   S700_1_WELD_BUFF_DATA5.RBT23_WELD_COUNT := W#16#0;
   S700_1_WELD_BUFF_DATA5.RBT24_BT_CODE_NO := W#16#0;
   S700_1_WELD_BUFF_DATA5.RBT24_WELD_COUNT := W#16#0;
   S700_1_WELD_BUFF_DATA5.WELD_DETERMINES_RESULT := W#16#0;
   S700_1_WELD_BUFF_DATA5.WELD_CHECK_SUM := W#16#0;
   S700_1_WELD_BUFF_DATA5.SPARE1 := W#16#0;
   S700_1_WELD_BUFF_DATA6.STATION_MAIN := W#16#0;
   S700_1_WELD_BUFF_DATA6.DISTINCTION_LH_RH := W#16#0;
   S700_1_WELD_BUFF_DATA6.STAION_NUMBER := W#16#0;
   S700_1_WELD_BUFF_DATA6.VIN_NUMBER1 := W#16#0;
   S700_1_WELD_BUFF_DATA6.VIN_NUMBER2 := W#16#0;
   S700_1_WELD_BUFF_DATA6.VIN_NUMBER3 := W#16#0;
   S700_1_WELD_BUFF_DATA6.VIN_NUMBER4 := W#16#0;
   S700_1_WELD_BUFF_DATA6.SEQ_NUMBER1 := W#16#0;
   S700_1_WELD_BUFF_DATA6.SEQ_NUMBER2 := W#16#0;
   S700_1_WELD_BUFF_DATA6.RBT1_BT_CODE_NO := W#16#0;
   S700_1_WELD_BUFF_DATA6.RBT1_WELD_COUNT := W#16#0;
   S700_1_WELD_BUFF_DATA6.RBT2_BT_CODE_NO := W#16#0;
   S700_1_WELD_BUFF_DATA6.RBT2_WELD_COUNT := W#16#0;
   S700_1_WELD_BUFF_DATA6.RBT3_BT_CODE_NO := W#16#0;
   S700_1_WELD_BUFF_DATA6.RBT3_WELD_COUNT := W#16#0;
   S700_1_WELD_BUFF_DATA6.RBT4_BT_CODE_NO := W#16#0;
   S700_1_WELD_BUFF_DATA6.RBT4_WELD_COUNT := W#16#0;
   S700_1_WELD_BUFF_DATA6.RBT5_BT_CODE_NO := W#16#0;
   S700_1_WELD_BUFF_DATA6.RBT5_WELD_COUNT := W#16#0;
   S700_1_WELD_BUFF_DATA6.RBT6_BT_CODE_NO := W#16#0;
   S700_1_WELD_BUFF_DATA6.RBT6_WELD_COUNT := W#16#0;
   S700_1_WELD_BUFF_DATA6.RBT7_BT_CODE_NO := W#16#0;
   S700_1_WELD_BUFF_DATA6.RBT7_WELD_COUNT := W#16#0;
   S700_1_WELD_BUFF_DATA6.RBT8_BT_CODE_NO := W#16#0;
   S700_1_WELD_BUFF_DATA6.RBT8_WELD_COUNT := W#16#0;
   S700_1_WELD_BUFF_DATA6.RBT9_BT_CODE_NO := W#16#0;
   S700_1_WELD_BUFF_DATA6.RBT9_WELD_COUNT := W#16#0;
   S700_1_WELD_BUFF_DATA6.RBT10_BT_CODE_NO := W#16#0;
   S700_1_WELD_BUFF_DATA6.RBT10_WELD_COUNT := W#16#0;
   S700_1_WELD_BUFF_DATA6.RBT11_BT_CODE_NO := W#16#0;
   S700_1_WELD_BUFF_DATA6.RBT11_WELD_COUNT := W#16#0;
   S700_1_WELD_BUFF_DATA6.RBT12_BT_CODE_NO := W#16#0;
   S700_1_WELD_BUFF_DATA6.RBT12_WELD_COUNT := W#16#0;
   S700_1_WELD_BUFF_DATA6.RBT13_BT_CODE_NO := W#16#0;
   S700_1_WELD_BUFF_DATA6.RBT13_WELD_COUNT := W#16#0;
   S700_1_WELD_BUFF_DATA6.RBT14_BT_CODE_NO := W#16#0;
   S700_1_WELD_BUFF_DATA6.RBT14_WELD_COUNT := W#16#0;
   S700_1_WELD_BUFF_DATA6.RBT15_BT_CODE_NO := W#16#0;
   S700_1_WELD_BUFF_DATA6.RBT15_WELD_COUNT := W#16#0;
   S700_1_WELD_BUFF_DATA6.RBT16_BT_CODE_NO := W#16#0;
   S700_1_WELD_BUFF_DATA6.RBT16_WELD_COUNT := W#16#0;
   S700_1_WELD_BUFF_DATA6.RBT17_BT_CODE_NO := W#16#0;
   S700_1_WELD_BUFF_DATA6.RBT17_WELD_COUNT := W#16#0;
   S700_1_WELD_BUFF_DATA6.RBT18_BT_CODE_NO := W#16#0;
   S700_1_WELD_BUFF_DATA6.RBT18_WELD_COUNT := W#16#0;
   S700_1_WELD_BUFF_DATA6.RBT19_BT_CODE_NO := W#16#0;
   S700_1_WELD_BUFF_DATA6.RBT19_WELD_COUNT := W#16#0;
   S700_1_WELD_BUFF_DATA6.RBT20_BT_CODE_NO := W#16#0;
   S700_1_WELD_BUFF_DATA6.RBT20_WELD_COUNT := W#16#0;
   S700_1_WELD_BUFF_DATA6.RBT21_BT_CODE_NO := W#16#0;
   S700_1_WELD_BUFF_DATA6.RBT21_WELD_COUNT := W#16#0;
   S700_1_WELD_BUFF_DATA6.RBT22_BT_CODE_NO := W#16#0;
   S700_1_WELD_BUFF_DATA6.RBT22_WELD_COUNT := W#16#0;
   S700_1_WELD_BUFF_DATA6.RBT23_BT_CODE_NO := W#16#0;
   S700_1_WELD_BUFF_DATA6.RBT23_WELD_COUNT := W#16#0;
   S700_1_WELD_BUFF_DATA6.RBT24_BT_CODE_NO := W#16#0;
   S700_1_WELD_BUFF_DATA6.RBT24_WELD_COUNT := W#16#0;
   S700_1_WELD_BUFF_DATA6.WELD_DETERMINES_RESULT := W#16#0;
   S700_1_WELD_BUFF_DATA6.WELD_CHECK_SUM := W#16#0;
   S700_1_WELD_BUFF_DATA6.SPARE1 := W#16#0;
   S700_1_WELD_BUFF_DATA7.STATION_MAIN := W#16#0;
   S700_1_WELD_BUFF_DATA7.DISTINCTION_LH_RH := W#16#0;
   S700_1_WELD_BUFF_DATA7.STAION_NUMBER := W#16#0;
   S700_1_WELD_BUFF_DATA7.VIN_NUMBER1 := W#16#0;
   S700_1_WELD_BUFF_DATA7.VIN_NUMBER2 := W#16#0;
   S700_1_WELD_BUFF_DATA7.VIN_NUMBER3 := W#16#0;
   S700_1_WELD_BUFF_DATA7.VIN_NUMBER4 := W#16#0;
   S700_1_WELD_BUFF_DATA7.SEQ_NUMBER1 := W#16#0;
   S700_1_WELD_BUFF_DATA7.SEQ_NUMBER2 := W#16#0;
   S700_1_WELD_BUFF_DATA7.RBT1_BT_CODE_NO := W#16#0;
   S700_1_WELD_BUFF_DATA7.RBT1_WELD_COUNT := W#16#0;
   S700_1_WELD_BUFF_DATA7.RBT2_BT_CODE_NO := W#16#0;
   S700_1_WELD_BUFF_DATA7.RBT2_WELD_COUNT := W#16#0;
   S700_1_WELD_BUFF_DATA7.RBT3_BT_CODE_NO := W#16#0;
   S700_1_WELD_BUFF_DATA7.RBT3_WELD_COUNT := W#16#0;
   S700_1_WELD_BUFF_DATA7.RBT4_BT_CODE_NO := W#16#0;
   S700_1_WELD_BUFF_DATA7.RBT4_WELD_COUNT := W#16#0;
   S700_1_WELD_BUFF_DATA7.RBT5_BT_CODE_NO := W#16#0;
   S700_1_WELD_BUFF_DATA7.RBT5_WELD_COUNT := W#16#0;
   S700_1_WELD_BUFF_DATA7.RBT6_BT_CODE_NO := W#16#0;
   S700_1_WELD_BUFF_DATA7.RBT6_WELD_COUNT := W#16#0;
   S700_1_WELD_BUFF_DATA7.RBT7_BT_CODE_NO := W#16#0;
   S700_1_WELD_BUFF_DATA7.RBT7_WELD_COUNT := W#16#0;
   S700_1_WELD_BUFF_DATA7.RBT8_BT_CODE_NO := W#16#0;
   S700_1_WELD_BUFF_DATA7.RBT8_WELD_COUNT := W#16#0;
   S700_1_WELD_BUFF_DATA7.RBT9_BT_CODE_NO := W#16#0;
   S700_1_WELD_BUFF_DATA7.RBT9_WELD_COUNT := W#16#0;
   S700_1_WELD_BUFF_DATA7.RBT10_BT_CODE_NO := W#16#0;
   S700_1_WELD_BUFF_DATA7.RBT10_WELD_COUNT := W#16#0;
   S700_1_WELD_BUFF_DATA7.RBT11_BT_CODE_NO := W#16#0;
   S700_1_WELD_BUFF_DATA7.RBT11_WELD_COUNT := W#16#0;
   S700_1_WELD_BUFF_DATA7.RBT12_BT_CODE_NO := W#16#0;
   S700_1_WELD_BUFF_DATA7.RBT12_WELD_COUNT := W#16#0;
   S700_1_WELD_BUFF_DATA7.RBT13_BT_CODE_NO := W#16#0;
   S700_1_WELD_BUFF_DATA7.RBT13_WELD_COUNT := W#16#0;
   S700_1_WELD_BUFF_DATA7.RBT14_BT_CODE_NO := W#16#0;
   S700_1_WELD_BUFF_DATA7.RBT14_WELD_COUNT := W#16#0;
   S700_1_WELD_BUFF_DATA7.RBT15_BT_CODE_NO := W#16#0;
   S700_1_WELD_BUFF_DATA7.RBT15_WELD_COUNT := W#16#0;
   S700_1_WELD_BUFF_DATA7.RBT16_BT_CODE_NO := W#16#0;
   S700_1_WELD_BUFF_DATA7.RBT16_WELD_COUNT := W#16#0;
   S700_1_WELD_BUFF_DATA7.RBT17_BT_CODE_NO := W#16#0;
   S700_1_WELD_BUFF_DATA7.RBT17_WELD_COUNT := W#16#0;
   S700_1_WELD_BUFF_DATA7.RBT18_BT_CODE_NO := W#16#0;
   S700_1_WELD_BUFF_DATA7.RBT18_WELD_COUNT := W#16#0;
   S700_1_WELD_BUFF_DATA7.RBT19_BT_CODE_NO := W#16#0;
   S700_1_WELD_BUFF_DATA7.RBT19_WELD_COUNT := W#16#0;
   S700_1_WELD_BUFF_DATA7.RBT20_BT_CODE_NO := W#16#0;
   S700_1_WELD_BUFF_DATA7.RBT20_WELD_COUNT := W#16#0;
   S700_1_WELD_BUFF_DATA7.RBT21_BT_CODE_NO := W#16#0;
   S700_1_WELD_BUFF_DATA7.RBT21_WELD_COUNT := W#16#0;
   S700_1_WELD_BUFF_DATA7.RBT22_BT_CODE_NO := W#16#0;
   S700_1_WELD_BUFF_DATA7.RBT22_WELD_COUNT := W#16#0;
   S700_1_WELD_BUFF_DATA7.RBT23_BT_CODE_NO := W#16#0;
   S700_1_WELD_BUFF_DATA7.RBT23_WELD_COUNT := W#16#0;
   S700_1_WELD_BUFF_DATA7.RBT24_BT_CODE_NO := W#16#0;
   S700_1_WELD_BUFF_DATA7.RBT24_WELD_COUNT := W#16#0;
   S700_1_WELD_BUFF_DATA7.WELD_DETERMINES_RESULT := W#16#0;
   S700_1_WELD_BUFF_DATA7.WELD_CHECK_SUM := W#16#0;
   S700_1_WELD_BUFF_DATA7.SPARE1 := W#16#0;
   S700_1_WELD_BUFF_DATA8.STATION_MAIN := W#16#0;
   S700_1_WELD_BUFF_DATA8.DISTINCTION_LH_RH := W#16#0;
   S700_1_WELD_BUFF_DATA8.STAION_NUMBER := W#16#0;
   S700_1_WELD_BUFF_DATA8.VIN_NUMBER1 := W#16#0;
   S700_1_WELD_BUFF_DATA8.VIN_NUMBER2 := W#16#0;
   S700_1_WELD_BUFF_DATA8.VIN_NUMBER3 := W#16#0;
   S700_1_WELD_BUFF_DATA8.VIN_NUMBER4 := W#16#0;
   S700_1_WELD_BUFF_DATA8.SEQ_NUMBER1 := W#16#0;
   S700_1_WELD_BUFF_DATA8.SEQ_NUMBER2 := W#16#0;
   S700_1_WELD_BUFF_DATA8.RBT1_BT_CODE_NO := W#16#0;
   S700_1_WELD_BUFF_DATA8.RBT1_WELD_COUNT := W#16#0;
   S700_1_WELD_BUFF_DATA8.RBT2_BT_CODE_NO := W#16#0;
   S700_1_WELD_BUFF_DATA8.RBT2_WELD_COUNT := W#16#0;
   S700_1_WELD_BUFF_DATA8.RBT3_BT_CODE_NO := W#16#0;
   S700_1_WELD_BUFF_DATA8.RBT3_WELD_COUNT := W#16#0;
   S700_1_WELD_BUFF_DATA8.RBT4_BT_CODE_NO := W#16#0;
   S700_1_WELD_BUFF_DATA8.RBT4_WELD_COUNT := W#16#0;
   S700_1_WELD_BUFF_DATA8.RBT5_BT_CODE_NO := W#16#0;
   S700_1_WELD_BUFF_DATA8.RBT5_WELD_COUNT := W#16#0;
   S700_1_WELD_BUFF_DATA8.RBT6_BT_CODE_NO := W#16#0;
   S700_1_WELD_BUFF_DATA8.RBT6_WELD_COUNT := W#16#0;
   S700_1_WELD_BUFF_DATA8.RBT7_BT_CODE_NO := W#16#0;
   S700_1_WELD_BUFF_DATA8.RBT7_WELD_COUNT := W#16#0;
   S700_1_WELD_BUFF_DATA8.RBT8_BT_CODE_NO := W#16#0;
   S700_1_WELD_BUFF_DATA8.RBT8_WELD_COUNT := W#16#0;
   S700_1_WELD_BUFF_DATA8.RBT9_BT_CODE_NO := W#16#0;
   S700_1_WELD_BUFF_DATA8.RBT9_WELD_COUNT := W#16#0;
   S700_1_WELD_BUFF_DATA8.RBT10_BT_CODE_NO := W#16#0;
   S700_1_WELD_BUFF_DATA8.RBT10_WELD_COUNT := W#16#0;
   S700_1_WELD_BUFF_DATA8.RBT11_BT_CODE_NO := W#16#0;
   S700_1_WELD_BUFF_DATA8.RBT11_WELD_COUNT := W#16#0;
   S700_1_WELD_BUFF_DATA8.RBT12_BT_CODE_NO := W#16#0;
   S700_1_WELD_BUFF_DATA8.RBT12_WELD_COUNT := W#16#0;
   S700_1_WELD_BUFF_DATA8.RBT13_BT_CODE_NO := W#16#0;
   S700_1_WELD_BUFF_DATA8.RBT13_WELD_COUNT := W#16#0;
   S700_1_WELD_BUFF_DATA8.RBT14_BT_CODE_NO := W#16#0;
   S700_1_WELD_BUFF_DATA8.RBT14_WELD_COUNT := W#16#0;
   S700_1_WELD_BUFF_DATA8.RBT15_BT_CODE_NO := W#16#0;
   S700_1_WELD_BUFF_DATA8.RBT15_WELD_COUNT := W#16#0;
   S700_1_WELD_BUFF_DATA8.RBT16_BT_CODE_NO := W#16#0;
   S700_1_WELD_BUFF_DATA8.RBT16_WELD_COUNT := W#16#0;
   S700_1_WELD_BUFF_DATA8.RBT17_BT_CODE_NO := W#16#0;
   S700_1_WELD_BUFF_DATA8.RBT17_WELD_COUNT := W#16#0;
   S700_1_WELD_BUFF_DATA8.RBT18_BT_CODE_NO := W#16#0;
   S700_1_WELD_BUFF_DATA8.RBT18_WELD_COUNT := W#16#0;
   S700_1_WELD_BUFF_DATA8.RBT19_BT_CODE_NO := W#16#0;
   S700_1_WELD_BUFF_DATA8.RBT19_WELD_COUNT := W#16#0;
   S700_1_WELD_BUFF_DATA8.RBT20_BT_CODE_NO := W#16#0;
   S700_1_WELD_BUFF_DATA8.RBT20_WELD_COUNT := W#16#0;
   S700_1_WELD_BUFF_DATA8.RBT21_BT_CODE_NO := W#16#0;
   S700_1_WELD_BUFF_DATA8.RBT21_WELD_COUNT := W#16#0;
   S700_1_WELD_BUFF_DATA8.RBT22_BT_CODE_NO := W#16#0;
   S700_1_WELD_BUFF_DATA8.RBT22_WELD_COUNT := W#16#0;
   S700_1_WELD_BUFF_DATA8.RBT23_BT_CODE_NO := W#16#0;
   S700_1_WELD_BUFF_DATA8.RBT23_WELD_COUNT := W#16#0;
   S700_1_WELD_BUFF_DATA8.RBT24_BT_CODE_NO := W#16#0;
   S700_1_WELD_BUFF_DATA8.RBT24_WELD_COUNT := W#16#0;
   S700_1_WELD_BUFF_DATA8.WELD_DETERMINES_RESULT := W#16#0;
   S700_1_WELD_BUFF_DATA8.WELD_CHECK_SUM := W#16#0;
   S700_1_WELD_BUFF_DATA8.SPARE1 := W#16#0;
   S700_1_WELD_BUFF_DATA9.STATION_MAIN := W#16#0;
   S700_1_WELD_BUFF_DATA9.DISTINCTION_LH_RH := W#16#0;
   S700_1_WELD_BUFF_DATA9.STAION_NUMBER := W#16#0;
   S700_1_WELD_BUFF_DATA9.VIN_NUMBER1 := W#16#0;
   S700_1_WELD_BUFF_DATA9.VIN_NUMBER2 := W#16#0;
   S700_1_WELD_BUFF_DATA9.VIN_NUMBER3 := W#16#0;
   S700_1_WELD_BUFF_DATA9.VIN_NUMBER4 := W#16#0;
   S700_1_WELD_BUFF_DATA9.SEQ_NUMBER1 := W#16#0;
   S700_1_WELD_BUFF_DATA9.SEQ_NUMBER2 := W#16#0;
   S700_1_WELD_BUFF_DATA9.RBT1_BT_CODE_NO := W#16#0;
   S700_1_WELD_BUFF_DATA9.RBT1_WELD_COUNT := W#16#0;
   S700_1_WELD_BUFF_DATA9.RBT2_BT_CODE_NO := W#16#0;
   S700_1_WELD_BUFF_DATA9.RBT2_WELD_COUNT := W#16#0;
   S700_1_WELD_BUFF_DATA9.RBT3_BT_CODE_NO := W#16#0;
   S700_1_WELD_BUFF_DATA9.RBT3_WELD_COUNT := W#16#0;
   S700_1_WELD_BUFF_DATA9.RBT4_BT_CODE_NO := W#16#0;
   S700_1_WELD_BUFF_DATA9.RBT4_WELD_COUNT := W#16#0;
   S700_1_WELD_BUFF_DATA9.RBT5_BT_CODE_NO := W#16#0;
   S700_1_WELD_BUFF_DATA9.RBT5_WELD_COUNT := W#16#0;
   S700_1_WELD_BUFF_DATA9.RBT6_BT_CODE_NO := W#16#0;
   S700_1_WELD_BUFF_DATA9.RBT6_WELD_COUNT := W#16#0;
   S700_1_WELD_BUFF_DATA9.RBT7_BT_CODE_NO := W#16#0;
   S700_1_WELD_BUFF_DATA9.RBT7_WELD_COUNT := W#16#0;
   S700_1_WELD_BUFF_DATA9.RBT8_BT_CODE_NO := W#16#0;
   S700_1_WELD_BUFF_DATA9.RBT8_WELD_COUNT := W#16#0;
   S700_1_WELD_BUFF_DATA9.RBT9_BT_CODE_NO := W#16#0;
   S700_1_WELD_BUFF_DATA9.RBT9_WELD_COUNT := W#16#0;
   S700_1_WELD_BUFF_DATA9.RBT10_BT_CODE_NO := W#16#0;
   S700_1_WELD_BUFF_DATA9.RBT10_WELD_COUNT := W#16#0;
   S700_1_WELD_BUFF_DATA9.RBT11_BT_CODE_NO := W#16#0;
   S700_1_WELD_BUFF_DATA9.RBT11_WELD_COUNT := W#16#0;
   S700_1_WELD_BUFF_DATA9.RBT12_BT_CODE_NO := W#16#0;
   S700_1_WELD_BUFF_DATA9.RBT12_WELD_COUNT := W#16#0;
   S700_1_WELD_BUFF_DATA9.RBT13_BT_CODE_NO := W#16#0;
   S700_1_WELD_BUFF_DATA9.RBT13_WELD_COUNT := W#16#0;
   S700_1_WELD_BUFF_DATA9.RBT14_BT_CODE_NO := W#16#0;
   S700_1_WELD_BUFF_DATA9.RBT14_WELD_COUNT := W#16#0;
   S700_1_WELD_BUFF_DATA9.RBT15_BT_CODE_NO := W#16#0;
   S700_1_WELD_BUFF_DATA9.RBT15_WELD_COUNT := W#16#0;
   S700_1_WELD_BUFF_DATA9.RBT16_BT_CODE_NO := W#16#0;
   S700_1_WELD_BUFF_DATA9.RBT16_WELD_COUNT := W#16#0;
   S700_1_WELD_BUFF_DATA9.RBT17_BT_CODE_NO := W#16#0;
   S700_1_WELD_BUFF_DATA9.RBT17_WELD_COUNT := W#16#0;
   S700_1_WELD_BUFF_DATA9.RBT18_BT_CODE_NO := W#16#0;
   S700_1_WELD_BUFF_DATA9.RBT18_WELD_COUNT := W#16#0;
   S700_1_WELD_BUFF_DATA9.RBT19_BT_CODE_NO := W#16#0;
   S700_1_WELD_BUFF_DATA9.RBT19_WELD_COUNT := W#16#0;
   S700_1_WELD_BUFF_DATA9.RBT20_BT_CODE_NO := W#16#0;
   S700_1_WELD_BUFF_DATA9.RBT20_WELD_COUNT := W#16#0;
   S700_1_WELD_BUFF_DATA9.RBT21_BT_CODE_NO := W#16#0;
   S700_1_WELD_BUFF_DATA9.RBT21_WELD_COUNT := W#16#0;
   S700_1_WELD_BUFF_DATA9.RBT22_BT_CODE_NO := W#16#0;
   S700_1_WELD_BUFF_DATA9.RBT22_WELD_COUNT := W#16#0;
   S700_1_WELD_BUFF_DATA9.RBT23_BT_CODE_NO := W#16#0;
   S700_1_WELD_BUFF_DATA9.RBT23_WELD_COUNT := W#16#0;
   S700_1_WELD_BUFF_DATA9.RBT24_BT_CODE_NO := W#16#0;
   S700_1_WELD_BUFF_DATA9.RBT24_WELD_COUNT := W#16#0;
   S700_1_WELD_BUFF_DATA9.WELD_DETERMINES_RESULT := W#16#0;
   S700_1_WELD_BUFF_DATA9.WELD_CHECK_SUM := W#16#0;
   S700_1_WELD_BUFF_DATA9.SPARE1 := W#16#0;
   S700_1_WELD_BUFF_DATA10.STATION_MAIN := W#16#0;
   S700_1_WELD_BUFF_DATA10.DISTINCTION_LH_RH := W#16#0;
   S700_1_WELD_BUFF_DATA10.STAION_NUMBER := W#16#0;
   S700_1_WELD_BUFF_DATA10.VIN_NUMBER1 := W#16#0;
   S700_1_WELD_BUFF_DATA10.VIN_NUMBER2 := W#16#0;
   S700_1_WELD_BUFF_DATA10.VIN_NUMBER3 := W#16#0;
   S700_1_WELD_BUFF_DATA10.VIN_NUMBER4 := W#16#0;
   S700_1_WELD_BUFF_DATA10.SEQ_NUMBER1 := W#16#0;
   S700_1_WELD_BUFF_DATA10.SEQ_NUMBER2 := W#16#0;
   S700_1_WELD_BUFF_DATA10.RBT1_BT_CODE_NO := W#16#0;
   S700_1_WELD_BUFF_DATA10.RBT1_WELD_COUNT := W#16#0;
   S700_1_WELD_BUFF_DATA10.RBT2_BT_CODE_NO := W#16#0;
   S700_1_WELD_BUFF_DATA10.RBT2_WELD_COUNT := W#16#0;
   S700_1_WELD_BUFF_DATA10.RBT3_BT_CODE_NO := W#16#0;
   S700_1_WELD_BUFF_DATA10.RBT3_WELD_COUNT := W#16#0;
   S700_1_WELD_BUFF_DATA10.RBT4_BT_CODE_NO := W#16#0;
   S700_1_WELD_BUFF_DATA10.RBT4_WELD_COUNT := W#16#0;
   S700_1_WELD_BUFF_DATA10.RBT5_BT_CODE_NO := W#16#0;
   S700_1_WELD_BUFF_DATA10.RBT5_WELD_COUNT := W#16#0;
   S700_1_WELD_BUFF_DATA10.RBT6_BT_CODE_NO := W#16#0;
   S700_1_WELD_BUFF_DATA10.RBT6_WELD_COUNT := W#16#0;
   S700_1_WELD_BUFF_DATA10.RBT7_BT_CODE_NO := W#16#0;
   S700_1_WELD_BUFF_DATA10.RBT7_WELD_COUNT := W#16#0;
   S700_1_WELD_BUFF_DATA10.RBT8_BT_CODE_NO := W#16#0;
   S700_1_WELD_BUFF_DATA10.RBT8_WELD_COUNT := W#16#0;
   S700_1_WELD_BUFF_DATA10.RBT9_BT_CODE_NO := W#16#0;
   S700_1_WELD_BUFF_DATA10.RBT9_WELD_COUNT := W#16#0;
   S700_1_WELD_BUFF_DATA10.RBT10_BT_CODE_NO := W#16#0;
   S700_1_WELD_BUFF_DATA10.RBT10_WELD_COUNT := W#16#0;
   S700_1_WELD_BUFF_DATA10.RBT11_BT_CODE_NO := W#16#0;
   S700_1_WELD_BUFF_DATA10.RBT11_WELD_COUNT := W#16#0;
   S700_1_WELD_BUFF_DATA10.RBT12_BT_CODE_NO := W#16#0;
   S700_1_WELD_BUFF_DATA10.RBT12_WELD_COUNT := W#16#0;
   S700_1_WELD_BUFF_DATA10.RBT13_BT_CODE_NO := W#16#0;
   S700_1_WELD_BUFF_DATA10.RBT13_WELD_COUNT := W#16#0;
   S700_1_WELD_BUFF_DATA10.RBT14_BT_CODE_NO := W#16#0;
   S700_1_WELD_BUFF_DATA10.RBT14_WELD_COUNT := W#16#0;
   S700_1_WELD_BUFF_DATA10.RBT15_BT_CODE_NO := W#16#0;
   S700_1_WELD_BUFF_DATA10.RBT15_WELD_COUNT := W#16#0;
   S700_1_WELD_BUFF_DATA10.RBT16_BT_CODE_NO := W#16#0;
   S700_1_WELD_BUFF_DATA10.RBT16_WELD_COUNT := W#16#0;
   S700_1_WELD_BUFF_DATA10.RBT17_BT_CODE_NO := W#16#0;
   S700_1_WELD_BUFF_DATA10.RBT17_WELD_COUNT := W#16#0;
   S700_1_WELD_BUFF_DATA10.RBT18_BT_CODE_NO := W#16#0;
   S700_1_WELD_BUFF_DATA10.RBT18_WELD_COUNT := W#16#0;
   S700_1_WELD_BUFF_DATA10.RBT19_BT_CODE_NO := W#16#0;
   S700_1_WELD_BUFF_DATA10.RBT19_WELD_COUNT := W#16#0;
   S700_1_WELD_BUFF_DATA10.RBT20_BT_CODE_NO := W#16#0;
   S700_1_WELD_BUFF_DATA10.RBT20_WELD_COUNT := W#16#0;
   S700_1_WELD_BUFF_DATA10.RBT21_BT_CODE_NO := W#16#0;
   S700_1_WELD_BUFF_DATA10.RBT21_WELD_COUNT := W#16#0;
   S700_1_WELD_BUFF_DATA10.RBT22_BT_CODE_NO := W#16#0;
   S700_1_WELD_BUFF_DATA10.RBT22_WELD_COUNT := W#16#0;
   S700_1_WELD_BUFF_DATA10.RBT23_BT_CODE_NO := W#16#0;
   S700_1_WELD_BUFF_DATA10.RBT23_WELD_COUNT := W#16#0;
   S700_1_WELD_BUFF_DATA10.RBT24_BT_CODE_NO := W#16#0;
   S700_1_WELD_BUFF_DATA10.RBT24_WELD_COUNT := W#16#0;
   S700_1_WELD_BUFF_DATA10.WELD_DETERMINES_RESULT := W#16#0;
   S700_1_WELD_BUFF_DATA10.WELD_CHECK_SUM := W#16#0;
   S700_1_WELD_BUFF_DATA10.SPARE1 := W#16#0;
   S701_WELD_BUFF_DATA1.STATION_MAIN := W#16#0;
   S701_WELD_BUFF_DATA1.DISTINCTION_LH_RH := W#16#0;
   S701_WELD_BUFF_DATA1.STAION_NUMBER := W#16#0;
   S701_WELD_BUFF_DATA1.VIN_NUMBER1 := W#16#0;
   S701_WELD_BUFF_DATA1.VIN_NUMBER2 := W#16#0;
   S701_WELD_BUFF_DATA1.VIN_NUMBER3 := W#16#0;
   S701_WELD_BUFF_DATA1.VIN_NUMBER4 := W#16#0;
   S701_WELD_BUFF_DATA1.SEQ_NUMBER1 := W#16#0;
   S701_WELD_BUFF_DATA1.SEQ_NUMBER2 := W#16#0;
   S701_WELD_BUFF_DATA1.RBT1_BT_CODE_NO := W#16#0;
   S701_WELD_BUFF_DATA1.RBT1_WELD_COUNT := W#16#0;
   S701_WELD_BUFF_DATA1.RBT2_BT_CODE_NO := W#16#0;
   S701_WELD_BUFF_DATA1.RBT2_WELD_COUNT := W#16#0;
   S701_WELD_BUFF_DATA1.RBT3_BT_CODE_NO := W#16#0;
   S701_WELD_BUFF_DATA1.RBT3_WELD_COUNT := W#16#0;
   S701_WELD_BUFF_DATA1.RBT4_BT_CODE_NO := W#16#0;
   S701_WELD_BUFF_DATA1.RBT4_WELD_COUNT := W#16#0;
   S701_WELD_BUFF_DATA1.RBT5_BT_CODE_NO := W#16#0;
   S701_WELD_BUFF_DATA1.RBT5_WELD_COUNT := W#16#0;
   S701_WELD_BUFF_DATA1.RBT6_BT_CODE_NO := W#16#0;
   S701_WELD_BUFF_DATA1.RBT6_WELD_COUNT := W#16#0;
   S701_WELD_BUFF_DATA1.RBT7_BT_CODE_NO := W#16#0;
   S701_WELD_BUFF_DATA1.RBT7_WELD_COUNT := W#16#0;
   S701_WELD_BUFF_DATA1.RBT8_BT_CODE_NO := W#16#0;
   S701_WELD_BUFF_DATA1.RBT8_WELD_COUNT := W#16#0;
   S701_WELD_BUFF_DATA1.RBT9_BT_CODE_NO := W#16#0;
   S701_WELD_BUFF_DATA1.RBT9_WELD_COUNT := W#16#0;
   S701_WELD_BUFF_DATA1.RBT10_BT_CODE_NO := W#16#0;
   S701_WELD_BUFF_DATA1.RBT10_WELD_COUNT := W#16#0;
   S701_WELD_BUFF_DATA1.RBT11_BT_CODE_NO := W#16#0;
   S701_WELD_BUFF_DATA1.RBT11_WELD_COUNT := W#16#0;
   S701_WELD_BUFF_DATA1.RBT12_BT_CODE_NO := W#16#0;
   S701_WELD_BUFF_DATA1.RBT12_WELD_COUNT := W#16#0;
   S701_WELD_BUFF_DATA1.RBT13_BT_CODE_NO := W#16#0;
   S701_WELD_BUFF_DATA1.RBT13_WELD_COUNT := W#16#0;
   S701_WELD_BUFF_DATA1.RBT14_BT_CODE_NO := W#16#0;
   S701_WELD_BUFF_DATA1.RBT14_WELD_COUNT := W#16#0;
   S701_WELD_BUFF_DATA1.RBT15_BT_CODE_NO := W#16#0;
   S701_WELD_BUFF_DATA1.RBT15_WELD_COUNT := W#16#0;
   S701_WELD_BUFF_DATA1.RBT16_BT_CODE_NO := W#16#0;
   S701_WELD_BUFF_DATA1.RBT16_WELD_COUNT := W#16#0;
   S701_WELD_BUFF_DATA1.RBT17_BT_CODE_NO := W#16#0;
   S701_WELD_BUFF_DATA1.RBT17_WELD_COUNT := W#16#0;
   S701_WELD_BUFF_DATA1.RBT18_BT_CODE_NO := W#16#0;
   S701_WELD_BUFF_DATA1.RBT18_WELD_COUNT := W#16#0;
   S701_WELD_BUFF_DATA1.RBT19_BT_CODE_NO := W#16#0;
   S701_WELD_BUFF_DATA1.RBT19_WELD_COUNT := W#16#0;
   S701_WELD_BUFF_DATA1.RBT20_BT_CODE_NO := W#16#0;
   S701_WELD_BUFF_DATA1.RBT20_WELD_COUNT := W#16#0;
   S701_WELD_BUFF_DATA1.RBT21_BT_CODE_NO := W#16#0;
   S701_WELD_BUFF_DATA1.RBT21_WELD_COUNT := W#16#0;
   S701_WELD_BUFF_DATA1.RBT22_BT_CODE_NO := W#16#0;
   S701_WELD_BUFF_DATA1.RBT22_WELD_COUNT := W#16#0;
   S701_WELD_BUFF_DATA1.RBT23_BT_CODE_NO := W#16#0;
   S701_WELD_BUFF_DATA1.RBT23_WELD_COUNT := W#16#0;
   S701_WELD_BUFF_DATA1.RBT24_BT_CODE_NO := W#16#0;
   S701_WELD_BUFF_DATA1.RBT24_WELD_COUNT := W#16#0;
   S701_WELD_BUFF_DATA1.WELD_DETERMINES_RESULT := W#16#0;
   S701_WELD_BUFF_DATA1.WELD_CHECK_SUM := W#16#0;
   S701_WELD_BUFF_DATA1.SPARE1 := W#16#0;
   S701_WELD_BUFF_DATA2.STATION_MAIN := W#16#0;
   S701_WELD_BUFF_DATA2.DISTINCTION_LH_RH := W#16#0;
   S701_WELD_BUFF_DATA2.STAION_NUMBER := W#16#0;
   S701_WELD_BUFF_DATA2.VIN_NUMBER1 := W#16#0;
   S701_WELD_BUFF_DATA2.VIN_NUMBER2 := W#16#0;
   S701_WELD_BUFF_DATA2.VIN_NUMBER3 := W#16#0;
   S701_WELD_BUFF_DATA2.VIN_NUMBER4 := W#16#0;
   S701_WELD_BUFF_DATA2.SEQ_NUMBER1 := W#16#0;
   S701_WELD_BUFF_DATA2.SEQ_NUMBER2 := W#16#0;
   S701_WELD_BUFF_DATA2.RBT1_BT_CODE_NO := W#16#0;
   S701_WELD_BUFF_DATA2.RBT1_WELD_COUNT := W#16#0;
   S701_WELD_BUFF_DATA2.RBT2_BT_CODE_NO := W#16#0;
   S701_WELD_BUFF_DATA2.RBT2_WELD_COUNT := W#16#0;
   S701_WELD_BUFF_DATA2.RBT3_BT_CODE_NO := W#16#0;
   S701_WELD_BUFF_DATA2.RBT3_WELD_COUNT := W#16#0;
   S701_WELD_BUFF_DATA2.RBT4_BT_CODE_NO := W#16#0;
   S701_WELD_BUFF_DATA2.RBT4_WELD_COUNT := W#16#0;
   S701_WELD_BUFF_DATA2.RBT5_BT_CODE_NO := W#16#0;
   S701_WELD_BUFF_DATA2.RBT5_WELD_COUNT := W#16#0;
   S701_WELD_BUFF_DATA2.RBT6_BT_CODE_NO := W#16#0;
   S701_WELD_BUFF_DATA2.RBT6_WELD_COUNT := W#16#0;
   S701_WELD_BUFF_DATA2.RBT7_BT_CODE_NO := W#16#0;
   S701_WELD_BUFF_DATA2.RBT7_WELD_COUNT := W#16#0;
   S701_WELD_BUFF_DATA2.RBT8_BT_CODE_NO := W#16#0;
   S701_WELD_BUFF_DATA2.RBT8_WELD_COUNT := W#16#0;
   S701_WELD_BUFF_DATA2.RBT9_BT_CODE_NO := W#16#0;
   S701_WELD_BUFF_DATA2.RBT9_WELD_COUNT := W#16#0;
   S701_WELD_BUFF_DATA2.RBT10_BT_CODE_NO := W#16#0;
   S701_WELD_BUFF_DATA2.RBT10_WELD_COUNT := W#16#0;
   S701_WELD_BUFF_DATA2.RBT11_BT_CODE_NO := W#16#0;
   S701_WELD_BUFF_DATA2.RBT11_WELD_COUNT := W#16#0;
   S701_WELD_BUFF_DATA2.RBT12_BT_CODE_NO := W#16#0;
   S701_WELD_BUFF_DATA2.RBT12_WELD_COUNT := W#16#0;
   S701_WELD_BUFF_DATA2.RBT13_BT_CODE_NO := W#16#0;
   S701_WELD_BUFF_DATA2.RBT13_WELD_COUNT := W#16#0;
   S701_WELD_BUFF_DATA2.RBT14_BT_CODE_NO := W#16#0;
   S701_WELD_BUFF_DATA2.RBT14_WELD_COUNT := W#16#0;
   S701_WELD_BUFF_DATA2.RBT15_BT_CODE_NO := W#16#0;
   S701_WELD_BUFF_DATA2.RBT15_WELD_COUNT := W#16#0;
   S701_WELD_BUFF_DATA2.RBT16_BT_CODE_NO := W#16#0;
   S701_WELD_BUFF_DATA2.RBT16_WELD_COUNT := W#16#0;
   S701_WELD_BUFF_DATA2.RBT17_BT_CODE_NO := W#16#0;
   S701_WELD_BUFF_DATA2.RBT17_WELD_COUNT := W#16#0;
   S701_WELD_BUFF_DATA2.RBT18_BT_CODE_NO := W#16#0;
   S701_WELD_BUFF_DATA2.RBT18_WELD_COUNT := W#16#0;
   S701_WELD_BUFF_DATA2.RBT19_BT_CODE_NO := W#16#0;
   S701_WELD_BUFF_DATA2.RBT19_WELD_COUNT := W#16#0;
   S701_WELD_BUFF_DATA2.RBT20_BT_CODE_NO := W#16#0;
   S701_WELD_BUFF_DATA2.RBT20_WELD_COUNT := W#16#0;
   S701_WELD_BUFF_DATA2.RBT21_BT_CODE_NO := W#16#0;
   S701_WELD_BUFF_DATA2.RBT21_WELD_COUNT := W#16#0;
   S701_WELD_BUFF_DATA2.RBT22_BT_CODE_NO := W#16#0;
   S701_WELD_BUFF_DATA2.RBT22_WELD_COUNT := W#16#0;
   S701_WELD_BUFF_DATA2.RBT23_BT_CODE_NO := W#16#0;
   S701_WELD_BUFF_DATA2.RBT23_WELD_COUNT := W#16#0;
   S701_WELD_BUFF_DATA2.RBT24_BT_CODE_NO := W#16#0;
   S701_WELD_BUFF_DATA2.RBT24_WELD_COUNT := W#16#0;
   S701_WELD_BUFF_DATA2.WELD_DETERMINES_RESULT := W#16#0;
   S701_WELD_BUFF_DATA2.WELD_CHECK_SUM := W#16#0;
   S701_WELD_BUFF_DATA2.SPARE1 := W#16#0;
   S701_WELD_BUFF_DATA3.STATION_MAIN := W#16#0;
   S701_WELD_BUFF_DATA3.DISTINCTION_LH_RH := W#16#0;
   S701_WELD_BUFF_DATA3.STAION_NUMBER := W#16#0;
   S701_WELD_BUFF_DATA3.VIN_NUMBER1 := W#16#0;
   S701_WELD_BUFF_DATA3.VIN_NUMBER2 := W#16#0;
   S701_WELD_BUFF_DATA3.VIN_NUMBER3 := W#16#0;
   S701_WELD_BUFF_DATA3.VIN_NUMBER4 := W#16#0;
   S701_WELD_BUFF_DATA3.SEQ_NUMBER1 := W#16#0;
   S701_WELD_BUFF_DATA3.SEQ_NUMBER2 := W#16#0;
   S701_WELD_BUFF_DATA3.RBT1_BT_CODE_NO := W#16#0;
   S701_WELD_BUFF_DATA3.RBT1_WELD_COUNT := W#16#0;
   S701_WELD_BUFF_DATA3.RBT2_BT_CODE_NO := W#16#0;
   S701_WELD_BUFF_DATA3.RBT2_WELD_COUNT := W#16#0;
   S701_WELD_BUFF_DATA3.RBT3_BT_CODE_NO := W#16#0;
   S701_WELD_BUFF_DATA3.RBT3_WELD_COUNT := W#16#0;
   S701_WELD_BUFF_DATA3.RBT4_BT_CODE_NO := W#16#0;
   S701_WELD_BUFF_DATA3.RBT4_WELD_COUNT := W#16#0;
   S701_WELD_BUFF_DATA3.RBT5_BT_CODE_NO := W#16#0;
   S701_WELD_BUFF_DATA3.RBT5_WELD_COUNT := W#16#0;
   S701_WELD_BUFF_DATA3.RBT6_BT_CODE_NO := W#16#0;
   S701_WELD_BUFF_DATA3.RBT6_WELD_COUNT := W#16#0;
   S701_WELD_BUFF_DATA3.RBT7_BT_CODE_NO := W#16#0;
   S701_WELD_BUFF_DATA3.RBT7_WELD_COUNT := W#16#0;
   S701_WELD_BUFF_DATA3.RBT8_BT_CODE_NO := W#16#0;
   S701_WELD_BUFF_DATA3.RBT8_WELD_COUNT := W#16#0;
   S701_WELD_BUFF_DATA3.RBT9_BT_CODE_NO := W#16#0;
   S701_WELD_BUFF_DATA3.RBT9_WELD_COUNT := W#16#0;
   S701_WELD_BUFF_DATA3.RBT10_BT_CODE_NO := W#16#0;
   S701_WELD_BUFF_DATA3.RBT10_WELD_COUNT := W#16#0;
   S701_WELD_BUFF_DATA3.RBT11_BT_CODE_NO := W#16#0;
   S701_WELD_BUFF_DATA3.RBT11_WELD_COUNT := W#16#0;
   S701_WELD_BUFF_DATA3.RBT12_BT_CODE_NO := W#16#0;
   S701_WELD_BUFF_DATA3.RBT12_WELD_COUNT := W#16#0;
   S701_WELD_BUFF_DATA3.RBT13_BT_CODE_NO := W#16#0;
   S701_WELD_BUFF_DATA3.RBT13_WELD_COUNT := W#16#0;
   S701_WELD_BUFF_DATA3.RBT14_BT_CODE_NO := W#16#0;
   S701_WELD_BUFF_DATA3.RBT14_WELD_COUNT := W#16#0;
   S701_WELD_BUFF_DATA3.RBT15_BT_CODE_NO := W#16#0;
   S701_WELD_BUFF_DATA3.RBT15_WELD_COUNT := W#16#0;
   S701_WELD_BUFF_DATA3.RBT16_BT_CODE_NO := W#16#0;
   S701_WELD_BUFF_DATA3.RBT16_WELD_COUNT := W#16#0;
   S701_WELD_BUFF_DATA3.RBT17_BT_CODE_NO := W#16#0;
   S701_WELD_BUFF_DATA3.RBT17_WELD_COUNT := W#16#0;
   S701_WELD_BUFF_DATA3.RBT18_BT_CODE_NO := W#16#0;
   S701_WELD_BUFF_DATA3.RBT18_WELD_COUNT := W#16#0;
   S701_WELD_BUFF_DATA3.RBT19_BT_CODE_NO := W#16#0;
   S701_WELD_BUFF_DATA3.RBT19_WELD_COUNT := W#16#0;
   S701_WELD_BUFF_DATA3.RBT20_BT_CODE_NO := W#16#0;
   S701_WELD_BUFF_DATA3.RBT20_WELD_COUNT := W#16#0;
   S701_WELD_BUFF_DATA3.RBT21_BT_CODE_NO := W#16#0;
   S701_WELD_BUFF_DATA3.RBT21_WELD_COUNT := W#16#0;
   S701_WELD_BUFF_DATA3.RBT22_BT_CODE_NO := W#16#0;
   S701_WELD_BUFF_DATA3.RBT22_WELD_COUNT := W#16#0;
   S701_WELD_BUFF_DATA3.RBT23_BT_CODE_NO := W#16#0;
   S701_WELD_BUFF_DATA3.RBT23_WELD_COUNT := W#16#0;
   S701_WELD_BUFF_DATA3.RBT24_BT_CODE_NO := W#16#0;
   S701_WELD_BUFF_DATA3.RBT24_WELD_COUNT := W#16#0;
   S701_WELD_BUFF_DATA3.WELD_DETERMINES_RESULT := W#16#0;
   S701_WELD_BUFF_DATA3.WELD_CHECK_SUM := W#16#0;
   S701_WELD_BUFF_DATA3.SPARE1 := W#16#0;
   S701_WELD_BUFF_DATA4.STATION_MAIN := W#16#0;
   S701_WELD_BUFF_DATA4.DISTINCTION_LH_RH := W#16#0;
   S701_WELD_BUFF_DATA4.STAION_NUMBER := W#16#0;
   S701_WELD_BUFF_DATA4.VIN_NUMBER1 := W#16#0;
   S701_WELD_BUFF_DATA4.VIN_NUMBER2 := W#16#0;
   S701_WELD_BUFF_DATA4.VIN_NUMBER3 := W#16#0;
   S701_WELD_BUFF_DATA4.VIN_NUMBER4 := W#16#0;
   S701_WELD_BUFF_DATA4.SEQ_NUMBER1 := W#16#0;
   S701_WELD_BUFF_DATA4.SEQ_NUMBER2 := W#16#0;
   S701_WELD_BUFF_DATA4.RBT1_BT_CODE_NO := W#16#0;
   S701_WELD_BUFF_DATA4.RBT1_WELD_COUNT := W#16#0;
   S701_WELD_BUFF_DATA4.RBT2_BT_CODE_NO := W#16#0;
   S701_WELD_BUFF_DATA4.RBT2_WELD_COUNT := W#16#0;
   S701_WELD_BUFF_DATA4.RBT3_BT_CODE_NO := W#16#0;
   S701_WELD_BUFF_DATA4.RBT3_WELD_COUNT := W#16#0;
   S701_WELD_BUFF_DATA4.RBT4_BT_CODE_NO := W#16#0;
   S701_WELD_BUFF_DATA4.RBT4_WELD_COUNT := W#16#0;
   S701_WELD_BUFF_DATA4.RBT5_BT_CODE_NO := W#16#0;
   S701_WELD_BUFF_DATA4.RBT5_WELD_COUNT := W#16#0;
   S701_WELD_BUFF_DATA4.RBT6_BT_CODE_NO := W#16#0;
   S701_WELD_BUFF_DATA4.RBT6_WELD_COUNT := W#16#0;
   S701_WELD_BUFF_DATA4.RBT7_BT_CODE_NO := W#16#0;
   S701_WELD_BUFF_DATA4.RBT7_WELD_COUNT := W#16#0;
   S701_WELD_BUFF_DATA4.RBT8_BT_CODE_NO := W#16#0;
   S701_WELD_BUFF_DATA4.RBT8_WELD_COUNT := W#16#0;
   S701_WELD_BUFF_DATA4.RBT9_BT_CODE_NO := W#16#0;
   S701_WELD_BUFF_DATA4.RBT9_WELD_COUNT := W#16#0;
   S701_WELD_BUFF_DATA4.RBT10_BT_CODE_NO := W#16#0;
   S701_WELD_BUFF_DATA4.RBT10_WELD_COUNT := W#16#0;
   S701_WELD_BUFF_DATA4.RBT11_BT_CODE_NO := W#16#0;
   S701_WELD_BUFF_DATA4.RBT11_WELD_COUNT := W#16#0;
   S701_WELD_BUFF_DATA4.RBT12_BT_CODE_NO := W#16#0;
   S701_WELD_BUFF_DATA4.RBT12_WELD_COUNT := W#16#0;
   S701_WELD_BUFF_DATA4.RBT13_BT_CODE_NO := W#16#0;
   S701_WELD_BUFF_DATA4.RBT13_WELD_COUNT := W#16#0;
   S701_WELD_BUFF_DATA4.RBT14_BT_CODE_NO := W#16#0;
   S701_WELD_BUFF_DATA4.RBT14_WELD_COUNT := W#16#0;
   S701_WELD_BUFF_DATA4.RBT15_BT_CODE_NO := W#16#0;
   S701_WELD_BUFF_DATA4.RBT15_WELD_COUNT := W#16#0;
   S701_WELD_BUFF_DATA4.RBT16_BT_CODE_NO := W#16#0;
   S701_WELD_BUFF_DATA4.RBT16_WELD_COUNT := W#16#0;
   S701_WELD_BUFF_DATA4.RBT17_BT_CODE_NO := W#16#0;
   S701_WELD_BUFF_DATA4.RBT17_WELD_COUNT := W#16#0;
   S701_WELD_BUFF_DATA4.RBT18_BT_CODE_NO := W#16#0;
   S701_WELD_BUFF_DATA4.RBT18_WELD_COUNT := W#16#0;
   S701_WELD_BUFF_DATA4.RBT19_BT_CODE_NO := W#16#0;
   S701_WELD_BUFF_DATA4.RBT19_WELD_COUNT := W#16#0;
   S701_WELD_BUFF_DATA4.RBT20_BT_CODE_NO := W#16#0;
   S701_WELD_BUFF_DATA4.RBT20_WELD_COUNT := W#16#0;
   S701_WELD_BUFF_DATA4.RBT21_BT_CODE_NO := W#16#0;
   S701_WELD_BUFF_DATA4.RBT21_WELD_COUNT := W#16#0;
   S701_WELD_BUFF_DATA4.RBT22_BT_CODE_NO := W#16#0;
   S701_WELD_BUFF_DATA4.RBT22_WELD_COUNT := W#16#0;
   S701_WELD_BUFF_DATA4.RBT23_BT_CODE_NO := W#16#0;
   S701_WELD_BUFF_DATA4.RBT23_WELD_COUNT := W#16#0;
   S701_WELD_BUFF_DATA4.RBT24_BT_CODE_NO := W#16#0;
   S701_WELD_BUFF_DATA4.RBT24_WELD_COUNT := W#16#0;
   S701_WELD_BUFF_DATA4.WELD_DETERMINES_RESULT := W#16#0;
   S701_WELD_BUFF_DATA4.WELD_CHECK_SUM := W#16#0;
   S701_WELD_BUFF_DATA4.SPARE1 := W#16#0;
   S701_WELD_BUFF_DATA5.STATION_MAIN := W#16#0;
   S701_WELD_BUFF_DATA5.DISTINCTION_LH_RH := W#16#0;
   S701_WELD_BUFF_DATA5.STAION_NUMBER := W#16#0;
   S701_WELD_BUFF_DATA5.VIN_NUMBER1 := W#16#0;
   S701_WELD_BUFF_DATA5.VIN_NUMBER2 := W#16#0;
   S701_WELD_BUFF_DATA5.VIN_NUMBER3 := W#16#0;
   S701_WELD_BUFF_DATA5.VIN_NUMBER4 := W#16#0;
   S701_WELD_BUFF_DATA5.SEQ_NUMBER1 := W#16#0;
   S701_WELD_BUFF_DATA5.SEQ_NUMBER2 := W#16#0;
   S701_WELD_BUFF_DATA5.RBT1_BT_CODE_NO := W#16#0;
   S701_WELD_BUFF_DATA5.RBT1_WELD_COUNT := W#16#0;
   S701_WELD_BUFF_DATA5.RBT2_BT_CODE_NO := W#16#0;
   S701_WELD_BUFF_DATA5.RBT2_WELD_COUNT := W#16#0;
   S701_WELD_BUFF_DATA5.RBT3_BT_CODE_NO := W#16#0;
   S701_WELD_BUFF_DATA5.RBT3_WELD_COUNT := W#16#0;
   S701_WELD_BUFF_DATA5.RBT4_BT_CODE_NO := W#16#0;
   S701_WELD_BUFF_DATA5.RBT4_WELD_COUNT := W#16#0;
   S701_WELD_BUFF_DATA5.RBT5_BT_CODE_NO := W#16#0;
   S701_WELD_BUFF_DATA5.RBT5_WELD_COUNT := W#16#0;
   S701_WELD_BUFF_DATA5.RBT6_BT_CODE_NO := W#16#0;
   S701_WELD_BUFF_DATA5.RBT6_WELD_COUNT := W#16#0;
   S701_WELD_BUFF_DATA5.RBT7_BT_CODE_NO := W#16#0;
   S701_WELD_BUFF_DATA5.RBT7_WELD_COUNT := W#16#0;
   S701_WELD_BUFF_DATA5.RBT8_BT_CODE_NO := W#16#0;
   S701_WELD_BUFF_DATA5.RBT8_WELD_COUNT := W#16#0;
   S701_WELD_BUFF_DATA5.RBT9_BT_CODE_NO := W#16#0;
   S701_WELD_BUFF_DATA5.RBT9_WELD_COUNT := W#16#0;
   S701_WELD_BUFF_DATA5.RBT10_BT_CODE_NO := W#16#0;
   S701_WELD_BUFF_DATA5.RBT10_WELD_COUNT := W#16#0;
   S701_WELD_BUFF_DATA5.RBT11_BT_CODE_NO := W#16#0;
   S701_WELD_BUFF_DATA5.RBT11_WELD_COUNT := W#16#0;
   S701_WELD_BUFF_DATA5.RBT12_BT_CODE_NO := W#16#0;
   S701_WELD_BUFF_DATA5.RBT12_WELD_COUNT := W#16#0;
   S701_WELD_BUFF_DATA5.RBT13_BT_CODE_NO := W#16#0;
   S701_WELD_BUFF_DATA5.RBT13_WELD_COUNT := W#16#0;
   S701_WELD_BUFF_DATA5.RBT14_BT_CODE_NO := W#16#0;
   S701_WELD_BUFF_DATA5.RBT14_WELD_COUNT := W#16#0;
   S701_WELD_BUFF_DATA5.RBT15_BT_CODE_NO := W#16#0;
   S701_WELD_BUFF_DATA5.RBT15_WELD_COUNT := W#16#0;
   S701_WELD_BUFF_DATA5.RBT16_BT_CODE_NO := W#16#0;
   S701_WELD_BUFF_DATA5.RBT16_WELD_COUNT := W#16#0;
   S701_WELD_BUFF_DATA5.RBT17_BT_CODE_NO := W#16#0;
   S701_WELD_BUFF_DATA5.RBT17_WELD_COUNT := W#16#0;
   S701_WELD_BUFF_DATA5.RBT18_BT_CODE_NO := W#16#0;
   S701_WELD_BUFF_DATA5.RBT18_WELD_COUNT := W#16#0;
   S701_WELD_BUFF_DATA5.RBT19_BT_CODE_NO := W#16#0;
   S701_WELD_BUFF_DATA5.RBT19_WELD_COUNT := W#16#0;
   S701_WELD_BUFF_DATA5.RBT20_BT_CODE_NO := W#16#0;
   S701_WELD_BUFF_DATA5.RBT20_WELD_COUNT := W#16#0;
   S701_WELD_BUFF_DATA5.RBT21_BT_CODE_NO := W#16#0;
   S701_WELD_BUFF_DATA5.RBT21_WELD_COUNT := W#16#0;
   S701_WELD_BUFF_DATA5.RBT22_BT_CODE_NO := W#16#0;
   S701_WELD_BUFF_DATA5.RBT22_WELD_COUNT := W#16#0;
   S701_WELD_BUFF_DATA5.RBT23_BT_CODE_NO := W#16#0;
   S701_WELD_BUFF_DATA5.RBT23_WELD_COUNT := W#16#0;
   S701_WELD_BUFF_DATA5.RBT24_BT_CODE_NO := W#16#0;
   S701_WELD_BUFF_DATA5.RBT24_WELD_COUNT := W#16#0;
   S701_WELD_BUFF_DATA5.WELD_DETERMINES_RESULT := W#16#0;
   S701_WELD_BUFF_DATA5.WELD_CHECK_SUM := W#16#0;
   S701_WELD_BUFF_DATA5.SPARE1 := W#16#0;
   S701_WELD_BUFF_DATA6.STATION_MAIN := W#16#0;
   S701_WELD_BUFF_DATA6.DISTINCTION_LH_RH := W#16#0;
   S701_WELD_BUFF_DATA6.STAION_NUMBER := W#16#0;
   S701_WELD_BUFF_DATA6.VIN_NUMBER1 := W#16#0;
   S701_WELD_BUFF_DATA6.VIN_NUMBER2 := W#16#0;
   S701_WELD_BUFF_DATA6.VIN_NUMBER3 := W#16#0;
   S701_WELD_BUFF_DATA6.VIN_NUMBER4 := W#16#0;
   S701_WELD_BUFF_DATA6.SEQ_NUMBER1 := W#16#0;
   S701_WELD_BUFF_DATA6.SEQ_NUMBER2 := W#16#0;
   S701_WELD_BUFF_DATA6.RBT1_BT_CODE_NO := W#16#0;
   S701_WELD_BUFF_DATA6.RBT1_WELD_COUNT := W#16#0;
   S701_WELD_BUFF_DATA6.RBT2_BT_CODE_NO := W#16#0;
   S701_WELD_BUFF_DATA6.RBT2_WELD_COUNT := W#16#0;
   S701_WELD_BUFF_DATA6.RBT3_BT_CODE_NO := W#16#0;
   S701_WELD_BUFF_DATA6.RBT3_WELD_COUNT := W#16#0;
   S701_WELD_BUFF_DATA6.RBT4_BT_CODE_NO := W#16#0;
   S701_WELD_BUFF_DATA6.RBT4_WELD_COUNT := W#16#0;
   S701_WELD_BUFF_DATA6.RBT5_BT_CODE_NO := W#16#0;
   S701_WELD_BUFF_DATA6.RBT5_WELD_COUNT := W#16#0;
   S701_WELD_BUFF_DATA6.RBT6_BT_CODE_NO := W#16#0;
   S701_WELD_BUFF_DATA6.RBT6_WELD_COUNT := W#16#0;
   S701_WELD_BUFF_DATA6.RBT7_BT_CODE_NO := W#16#0;
   S701_WELD_BUFF_DATA6.RBT7_WELD_COUNT := W#16#0;
   S701_WELD_BUFF_DATA6.RBT8_BT_CODE_NO := W#16#0;
   S701_WELD_BUFF_DATA6.RBT8_WELD_COUNT := W#16#0;
   S701_WELD_BUFF_DATA6.RBT9_BT_CODE_NO := W#16#0;
   S701_WELD_BUFF_DATA6.RBT9_WELD_COUNT := W#16#0;
   S701_WELD_BUFF_DATA6.RBT10_BT_CODE_NO := W#16#0;
   S701_WELD_BUFF_DATA6.RBT10_WELD_COUNT := W#16#0;
   S701_WELD_BUFF_DATA6.RBT11_BT_CODE_NO := W#16#0;
   S701_WELD_BUFF_DATA6.RBT11_WELD_COUNT := W#16#0;
   S701_WELD_BUFF_DATA6.RBT12_BT_CODE_NO := W#16#0;
   S701_WELD_BUFF_DATA6.RBT12_WELD_COUNT := W#16#0;
   S701_WELD_BUFF_DATA6.RBT13_BT_CODE_NO := W#16#0;
   S701_WELD_BUFF_DATA6.RBT13_WELD_COUNT := W#16#0;
   S701_WELD_BUFF_DATA6.RBT14_BT_CODE_NO := W#16#0;
   S701_WELD_BUFF_DATA6.RBT14_WELD_COUNT := W#16#0;
   S701_WELD_BUFF_DATA6.RBT15_BT_CODE_NO := W#16#0;
   S701_WELD_BUFF_DATA6.RBT15_WELD_COUNT := W#16#0;
   S701_WELD_BUFF_DATA6.RBT16_BT_CODE_NO := W#16#0;
   S701_WELD_BUFF_DATA6.RBT16_WELD_COUNT := W#16#0;
   S701_WELD_BUFF_DATA6.RBT17_BT_CODE_NO := W#16#0;
   S701_WELD_BUFF_DATA6.RBT17_WELD_COUNT := W#16#0;
   S701_WELD_BUFF_DATA6.RBT18_BT_CODE_NO := W#16#0;
   S701_WELD_BUFF_DATA6.RBT18_WELD_COUNT := W#16#0;
   S701_WELD_BUFF_DATA6.RBT19_BT_CODE_NO := W#16#0;
   S701_WELD_BUFF_DATA6.RBT19_WELD_COUNT := W#16#0;
   S701_WELD_BUFF_DATA6.RBT20_BT_CODE_NO := W#16#0;
   S701_WELD_BUFF_DATA6.RBT20_WELD_COUNT := W#16#0;
   S701_WELD_BUFF_DATA6.RBT21_BT_CODE_NO := W#16#0;
   S701_WELD_BUFF_DATA6.RBT21_WELD_COUNT := W#16#0;
   S701_WELD_BUFF_DATA6.RBT22_BT_CODE_NO := W#16#0;
   S701_WELD_BUFF_DATA6.RBT22_WELD_COUNT := W#16#0;
   S701_WELD_BUFF_DATA6.RBT23_BT_CODE_NO := W#16#0;
   S701_WELD_BUFF_DATA6.RBT23_WELD_COUNT := W#16#0;
   S701_WELD_BUFF_DATA6.RBT24_BT_CODE_NO := W#16#0;
   S701_WELD_BUFF_DATA6.RBT24_WELD_COUNT := W#16#0;
   S701_WELD_BUFF_DATA6.WELD_DETERMINES_RESULT := W#16#0;
   S701_WELD_BUFF_DATA6.WELD_CHECK_SUM := W#16#0;
   S701_WELD_BUFF_DATA6.SPARE1 := W#16#0;
   S701_WELD_BUFF_DATA7.STATION_MAIN := W#16#0;
   S701_WELD_BUFF_DATA7.DISTINCTION_LH_RH := W#16#0;
   S701_WELD_BUFF_DATA7.STAION_NUMBER := W#16#0;
   S701_WELD_BUFF_DATA7.VIN_NUMBER1 := W#16#0;
   S701_WELD_BUFF_DATA7.VIN_NUMBER2 := W#16#0;
   S701_WELD_BUFF_DATA7.VIN_NUMBER3 := W#16#0;
   S701_WELD_BUFF_DATA7.VIN_NUMBER4 := W#16#0;
   S701_WELD_BUFF_DATA7.SEQ_NUMBER1 := W#16#0;
   S701_WELD_BUFF_DATA7.SEQ_NUMBER2 := W#16#0;
   S701_WELD_BUFF_DATA7.RBT1_BT_CODE_NO := W#16#0;
   S701_WELD_BUFF_DATA7.RBT1_WELD_COUNT := W#16#0;
   S701_WELD_BUFF_DATA7.RBT2_BT_CODE_NO := W#16#0;
   S701_WELD_BUFF_DATA7.RBT2_WELD_COUNT := W#16#0;
   S701_WELD_BUFF_DATA7.RBT3_BT_CODE_NO := W#16#0;
   S701_WELD_BUFF_DATA7.RBT3_WELD_COUNT := W#16#0;
   S701_WELD_BUFF_DATA7.RBT4_BT_CODE_NO := W#16#0;
   S701_WELD_BUFF_DATA7.RBT4_WELD_COUNT := W#16#0;
   S701_WELD_BUFF_DATA7.RBT5_BT_CODE_NO := W#16#0;
   S701_WELD_BUFF_DATA7.RBT5_WELD_COUNT := W#16#0;
   S701_WELD_BUFF_DATA7.RBT6_BT_CODE_NO := W#16#0;
   S701_WELD_BUFF_DATA7.RBT6_WELD_COUNT := W#16#0;
   S701_WELD_BUFF_DATA7.RBT7_BT_CODE_NO := W#16#0;
   S701_WELD_BUFF_DATA7.RBT7_WELD_COUNT := W#16#0;
   S701_WELD_BUFF_DATA7.RBT8_BT_CODE_NO := W#16#0;
   S701_WELD_BUFF_DATA7.RBT8_WELD_COUNT := W#16#0;
   S701_WELD_BUFF_DATA7.RBT9_BT_CODE_NO := W#16#0;
   S701_WELD_BUFF_DATA7.RBT9_WELD_COUNT := W#16#0;
   S701_WELD_BUFF_DATA7.RBT10_BT_CODE_NO := W#16#0;
   S701_WELD_BUFF_DATA7.RBT10_WELD_COUNT := W#16#0;
   S701_WELD_BUFF_DATA7.RBT11_BT_CODE_NO := W#16#0;
   S701_WELD_BUFF_DATA7.RBT11_WELD_COUNT := W#16#0;
   S701_WELD_BUFF_DATA7.RBT12_BT_CODE_NO := W#16#0;
   S701_WELD_BUFF_DATA7.RBT12_WELD_COUNT := W#16#0;
   S701_WELD_BUFF_DATA7.RBT13_BT_CODE_NO := W#16#0;
   S701_WELD_BUFF_DATA7.RBT13_WELD_COUNT := W#16#0;
   S701_WELD_BUFF_DATA7.RBT14_BT_CODE_NO := W#16#0;
   S701_WELD_BUFF_DATA7.RBT14_WELD_COUNT := W#16#0;
   S701_WELD_BUFF_DATA7.RBT15_BT_CODE_NO := W#16#0;
   S701_WELD_BUFF_DATA7.RBT15_WELD_COUNT := W#16#0;
   S701_WELD_BUFF_DATA7.RBT16_BT_CODE_NO := W#16#0;
   S701_WELD_BUFF_DATA7.RBT16_WELD_COUNT := W#16#0;
   S701_WELD_BUFF_DATA7.RBT17_BT_CODE_NO := W#16#0;
   S701_WELD_BUFF_DATA7.RBT17_WELD_COUNT := W#16#0;
   S701_WELD_BUFF_DATA7.RBT18_BT_CODE_NO := W#16#0;
   S701_WELD_BUFF_DATA7.RBT18_WELD_COUNT := W#16#0;
   S701_WELD_BUFF_DATA7.RBT19_BT_CODE_NO := W#16#0;
   S701_WELD_BUFF_DATA7.RBT19_WELD_COUNT := W#16#0;
   S701_WELD_BUFF_DATA7.RBT20_BT_CODE_NO := W#16#0;
   S701_WELD_BUFF_DATA7.RBT20_WELD_COUNT := W#16#0;
   S701_WELD_BUFF_DATA7.RBT21_BT_CODE_NO := W#16#0;
   S701_WELD_BUFF_DATA7.RBT21_WELD_COUNT := W#16#0;
   S701_WELD_BUFF_DATA7.RBT22_BT_CODE_NO := W#16#0;
   S701_WELD_BUFF_DATA7.RBT22_WELD_COUNT := W#16#0;
   S701_WELD_BUFF_DATA7.RBT23_BT_CODE_NO := W#16#0;
   S701_WELD_BUFF_DATA7.RBT23_WELD_COUNT := W#16#0;
   S701_WELD_BUFF_DATA7.RBT24_BT_CODE_NO := W#16#0;
   S701_WELD_BUFF_DATA7.RBT24_WELD_COUNT := W#16#0;
   S701_WELD_BUFF_DATA7.WELD_DETERMINES_RESULT := W#16#0;
   S701_WELD_BUFF_DATA7.WELD_CHECK_SUM := W#16#0;
   S701_WELD_BUFF_DATA7.SPARE1 := W#16#0;
   S701_WELD_BUFF_DATA8.STATION_MAIN := W#16#0;
   S701_WELD_BUFF_DATA8.DISTINCTION_LH_RH := W#16#0;
   S701_WELD_BUFF_DATA8.STAION_NUMBER := W#16#0;
   S701_WELD_BUFF_DATA8.VIN_NUMBER1 := W#16#0;
   S701_WELD_BUFF_DATA8.VIN_NUMBER2 := W#16#0;
   S701_WELD_BUFF_DATA8.VIN_NUMBER3 := W#16#0;
   S701_WELD_BUFF_DATA8.VIN_NUMBER4 := W#16#0;
   S701_WELD_BUFF_DATA8.SEQ_NUMBER1 := W#16#0;
   S701_WELD_BUFF_DATA8.SEQ_NUMBER2 := W#16#0;
   S701_WELD_BUFF_DATA8.RBT1_BT_CODE_NO := W#16#0;
   S701_WELD_BUFF_DATA8.RBT1_WELD_COUNT := W#16#0;
   S701_WELD_BUFF_DATA8.RBT2_BT_CODE_NO := W#16#0;
   S701_WELD_BUFF_DATA8.RBT2_WELD_COUNT := W#16#0;
   S701_WELD_BUFF_DATA8.RBT3_BT_CODE_NO := W#16#0;
   S701_WELD_BUFF_DATA8.RBT3_WELD_COUNT := W#16#0;
   S701_WELD_BUFF_DATA8.RBT4_BT_CODE_NO := W#16#0;
   S701_WELD_BUFF_DATA8.RBT4_WELD_COUNT := W#16#0;
   S701_WELD_BUFF_DATA8.RBT5_BT_CODE_NO := W#16#0;
   S701_WELD_BUFF_DATA8.RBT5_WELD_COUNT := W#16#0;
   S701_WELD_BUFF_DATA8.RBT6_BT_CODE_NO := W#16#0;
   S701_WELD_BUFF_DATA8.RBT6_WELD_COUNT := W#16#0;
   S701_WELD_BUFF_DATA8.RBT7_BT_CODE_NO := W#16#0;
   S701_WELD_BUFF_DATA8.RBT7_WELD_COUNT := W#16#0;
   S701_WELD_BUFF_DATA8.RBT8_BT_CODE_NO := W#16#0;
   S701_WELD_BUFF_DATA8.RBT8_WELD_COUNT := W#16#0;
   S701_WELD_BUFF_DATA8.RBT9_BT_CODE_NO := W#16#0;
   S701_WELD_BUFF_DATA8.RBT9_WELD_COUNT := W#16#0;
   S701_WELD_BUFF_DATA8.RBT10_BT_CODE_NO := W#16#0;
   S701_WELD_BUFF_DATA8.RBT10_WELD_COUNT := W#16#0;
   S701_WELD_BUFF_DATA8.RBT11_BT_CODE_NO := W#16#0;
   S701_WELD_BUFF_DATA8.RBT11_WELD_COUNT := W#16#0;
   S701_WELD_BUFF_DATA8.RBT12_BT_CODE_NO := W#16#0;
   S701_WELD_BUFF_DATA8.RBT12_WELD_COUNT := W#16#0;
   S701_WELD_BUFF_DATA8.RBT13_BT_CODE_NO := W#16#0;
   S701_WELD_BUFF_DATA8.RBT13_WELD_COUNT := W#16#0;
   S701_WELD_BUFF_DATA8.RBT14_BT_CODE_NO := W#16#0;
   S701_WELD_BUFF_DATA8.RBT14_WELD_COUNT := W#16#0;
   S701_WELD_BUFF_DATA8.RBT15_BT_CODE_NO := W#16#0;
   S701_WELD_BUFF_DATA8.RBT15_WELD_COUNT := W#16#0;
   S701_WELD_BUFF_DATA8.RBT16_BT_CODE_NO := W#16#0;
   S701_WELD_BUFF_DATA8.RBT16_WELD_COUNT := W#16#0;
   S701_WELD_BUFF_DATA8.RBT17_BT_CODE_NO := W#16#0;
   S701_WELD_BUFF_DATA8.RBT17_WELD_COUNT := W#16#0;
   S701_WELD_BUFF_DATA8.RBT18_BT_CODE_NO := W#16#0;
   S701_WELD_BUFF_DATA8.RBT18_WELD_COUNT := W#16#0;
   S701_WELD_BUFF_DATA8.RBT19_BT_CODE_NO := W#16#0;
   S701_WELD_BUFF_DATA8.RBT19_WELD_COUNT := W#16#0;
   S701_WELD_BUFF_DATA8.RBT20_BT_CODE_NO := W#16#0;
   S701_WELD_BUFF_DATA8.RBT20_WELD_COUNT := W#16#0;
   S701_WELD_BUFF_DATA8.RBT21_BT_CODE_NO := W#16#0;
   S701_WELD_BUFF_DATA8.RBT21_WELD_COUNT := W#16#0;
   S701_WELD_BUFF_DATA8.RBT22_BT_CODE_NO := W#16#0;
   S701_WELD_BUFF_DATA8.RBT22_WELD_COUNT := W#16#0;
   S701_WELD_BUFF_DATA8.RBT23_BT_CODE_NO := W#16#0;
   S701_WELD_BUFF_DATA8.RBT23_WELD_COUNT := W#16#0;
   S701_WELD_BUFF_DATA8.RBT24_BT_CODE_NO := W#16#0;
   S701_WELD_BUFF_DATA8.RBT24_WELD_COUNT := W#16#0;
   S701_WELD_BUFF_DATA8.WELD_DETERMINES_RESULT := W#16#0;
   S701_WELD_BUFF_DATA8.WELD_CHECK_SUM := W#16#0;
   S701_WELD_BUFF_DATA8.SPARE1 := W#16#0;
   S701_WELD_BUFF_DATA9.STATION_MAIN := W#16#0;
   S701_WELD_BUFF_DATA9.DISTINCTION_LH_RH := W#16#0;
   S701_WELD_BUFF_DATA9.STAION_NUMBER := W#16#0;
   S701_WELD_BUFF_DATA9.VIN_NUMBER1 := W#16#0;
   S701_WELD_BUFF_DATA9.VIN_NUMBER2 := W#16#0;
   S701_WELD_BUFF_DATA9.VIN_NUMBER3 := W#16#0;
   S701_WELD_BUFF_DATA9.VIN_NUMBER4 := W#16#0;
   S701_WELD_BUFF_DATA9.SEQ_NUMBER1 := W#16#0;
   S701_WELD_BUFF_DATA9.SEQ_NUMBER2 := W#16#0;
   S701_WELD_BUFF_DATA9.RBT1_BT_CODE_NO := W#16#0;
   S701_WELD_BUFF_DATA9.RBT1_WELD_COUNT := W#16#0;
   S701_WELD_BUFF_DATA9.RBT2_BT_CODE_NO := W#16#0;
   S701_WELD_BUFF_DATA9.RBT2_WELD_COUNT := W#16#0;
   S701_WELD_BUFF_DATA9.RBT3_BT_CODE_NO := W#16#0;
   S701_WELD_BUFF_DATA9.RBT3_WELD_COUNT := W#16#0;
   S701_WELD_BUFF_DATA9.RBT4_BT_CODE_NO := W#16#0;
   S701_WELD_BUFF_DATA9.RBT4_WELD_COUNT := W#16#0;
   S701_WELD_BUFF_DATA9.RBT5_BT_CODE_NO := W#16#0;
   S701_WELD_BUFF_DATA9.RBT5_WELD_COUNT := W#16#0;
   S701_WELD_BUFF_DATA9.RBT6_BT_CODE_NO := W#16#0;
   S701_WELD_BUFF_DATA9.RBT6_WELD_COUNT := W#16#0;
   S701_WELD_BUFF_DATA9.RBT7_BT_CODE_NO := W#16#0;
   S701_WELD_BUFF_DATA9.RBT7_WELD_COUNT := W#16#0;
   S701_WELD_BUFF_DATA9.RBT8_BT_CODE_NO := W#16#0;
   S701_WELD_BUFF_DATA9.RBT8_WELD_COUNT := W#16#0;
   S701_WELD_BUFF_DATA9.RBT9_BT_CODE_NO := W#16#0;
   S701_WELD_BUFF_DATA9.RBT9_WELD_COUNT := W#16#0;
   S701_WELD_BUFF_DATA9.RBT10_BT_CODE_NO := W#16#0;
   S701_WELD_BUFF_DATA9.RBT10_WELD_COUNT := W#16#0;
   S701_WELD_BUFF_DATA9.RBT11_BT_CODE_NO := W#16#0;
   S701_WELD_BUFF_DATA9.RBT11_WELD_COUNT := W#16#0;
   S701_WELD_BUFF_DATA9.RBT12_BT_CODE_NO := W#16#0;
   S701_WELD_BUFF_DATA9.RBT12_WELD_COUNT := W#16#0;
   S701_WELD_BUFF_DATA9.RBT13_BT_CODE_NO := W#16#0;
   S701_WELD_BUFF_DATA9.RBT13_WELD_COUNT := W#16#0;
   S701_WELD_BUFF_DATA9.RBT14_BT_CODE_NO := W#16#0;
   S701_WELD_BUFF_DATA9.RBT14_WELD_COUNT := W#16#0;
   S701_WELD_BUFF_DATA9.RBT15_BT_CODE_NO := W#16#0;
   S701_WELD_BUFF_DATA9.RBT15_WELD_COUNT := W#16#0;
   S701_WELD_BUFF_DATA9.RBT16_BT_CODE_NO := W#16#0;
   S701_WELD_BUFF_DATA9.RBT16_WELD_COUNT := W#16#0;
   S701_WELD_BUFF_DATA9.RBT17_BT_CODE_NO := W#16#0;
   S701_WELD_BUFF_DATA9.RBT17_WELD_COUNT := W#16#0;
   S701_WELD_BUFF_DATA9.RBT18_BT_CODE_NO := W#16#0;
   S701_WELD_BUFF_DATA9.RBT18_WELD_COUNT := W#16#0;
   S701_WELD_BUFF_DATA9.RBT19_BT_CODE_NO := W#16#0;
   S701_WELD_BUFF_DATA9.RBT19_WELD_COUNT := W#16#0;
   S701_WELD_BUFF_DATA9.RBT20_BT_CODE_NO := W#16#0;
   S701_WELD_BUFF_DATA9.RBT20_WELD_COUNT := W#16#0;
   S701_WELD_BUFF_DATA9.RBT21_BT_CODE_NO := W#16#0;
   S701_WELD_BUFF_DATA9.RBT21_WELD_COUNT := W#16#0;
   S701_WELD_BUFF_DATA9.RBT22_BT_CODE_NO := W#16#0;
   S701_WELD_BUFF_DATA9.RBT22_WELD_COUNT := W#16#0;
   S701_WELD_BUFF_DATA9.RBT23_BT_CODE_NO := W#16#0;
   S701_WELD_BUFF_DATA9.RBT23_WELD_COUNT := W#16#0;
   S701_WELD_BUFF_DATA9.RBT24_BT_CODE_NO := W#16#0;
   S701_WELD_BUFF_DATA9.RBT24_WELD_COUNT := W#16#0;
   S701_WELD_BUFF_DATA9.WELD_DETERMINES_RESULT := W#16#0;
   S701_WELD_BUFF_DATA9.WELD_CHECK_SUM := W#16#0;
   S701_WELD_BUFF_DATA9.SPARE1 := W#16#0;
   S701_WELD_BUFF_DATA10.STATION_MAIN := W#16#0;
   S701_WELD_BUFF_DATA10.DISTINCTION_LH_RH := W#16#0;
   S701_WELD_BUFF_DATA10.STAION_NUMBER := W#16#0;
   S701_WELD_BUFF_DATA10.VIN_NUMBER1 := W#16#0;
   S701_WELD_BUFF_DATA10.VIN_NUMBER2 := W#16#0;
   S701_WELD_BUFF_DATA10.VIN_NUMBER3 := W#16#0;
   S701_WELD_BUFF_DATA10.VIN_NUMBER4 := W#16#0;
   S701_WELD_BUFF_DATA10.SEQ_NUMBER1 := W#16#0;
   S701_WELD_BUFF_DATA10.SEQ_NUMBER2 := W#16#0;
   S701_WELD_BUFF_DATA10.RBT1_BT_CODE_NO := W#16#0;
   S701_WELD_BUFF_DATA10.RBT1_WELD_COUNT := W#16#0;
   S701_WELD_BUFF_DATA10.RBT2_BT_CODE_NO := W#16#0;
   S701_WELD_BUFF_DATA10.RBT2_WELD_COUNT := W#16#0;
   S701_WELD_BUFF_DATA10.RBT3_BT_CODE_NO := W#16#0;
   S701_WELD_BUFF_DATA10.RBT3_WELD_COUNT := W#16#0;
   S701_WELD_BUFF_DATA10.RBT4_BT_CODE_NO := W#16#0;
   S701_WELD_BUFF_DATA10.RBT4_WELD_COUNT := W#16#0;
   S701_WELD_BUFF_DATA10.RBT5_BT_CODE_NO := W#16#0;
   S701_WELD_BUFF_DATA10.RBT5_WELD_COUNT := W#16#0;
   S701_WELD_BUFF_DATA10.RBT6_BT_CODE_NO := W#16#0;
   S701_WELD_BUFF_DATA10.RBT6_WELD_COUNT := W#16#0;
   S701_WELD_BUFF_DATA10.RBT7_BT_CODE_NO := W#16#0;
   S701_WELD_BUFF_DATA10.RBT7_WELD_COUNT := W#16#0;
   S701_WELD_BUFF_DATA10.RBT8_BT_CODE_NO := W#16#0;
   S701_WELD_BUFF_DATA10.RBT8_WELD_COUNT := W#16#0;
   S701_WELD_BUFF_DATA10.RBT9_BT_CODE_NO := W#16#0;
   S701_WELD_BUFF_DATA10.RBT9_WELD_COUNT := W#16#0;
   S701_WELD_BUFF_DATA10.RBT10_BT_CODE_NO := W#16#0;
   S701_WELD_BUFF_DATA10.RBT10_WELD_COUNT := W#16#0;
   S701_WELD_BUFF_DATA10.RBT11_BT_CODE_NO := W#16#0;
   S701_WELD_BUFF_DATA10.RBT11_WELD_COUNT := W#16#0;
   S701_WELD_BUFF_DATA10.RBT12_BT_CODE_NO := W#16#0;
   S701_WELD_BUFF_DATA10.RBT12_WELD_COUNT := W#16#0;
   S701_WELD_BUFF_DATA10.RBT13_BT_CODE_NO := W#16#0;
   S701_WELD_BUFF_DATA10.RBT13_WELD_COUNT := W#16#0;
   S701_WELD_BUFF_DATA10.RBT14_BT_CODE_NO := W#16#0;
   S701_WELD_BUFF_DATA10.RBT14_WELD_COUNT := W#16#0;
   S701_WELD_BUFF_DATA10.RBT15_BT_CODE_NO := W#16#0;
   S701_WELD_BUFF_DATA10.RBT15_WELD_COUNT := W#16#0;
   S701_WELD_BUFF_DATA10.RBT16_BT_CODE_NO := W#16#0;
   S701_WELD_BUFF_DATA10.RBT16_WELD_COUNT := W#16#0;
   S701_WELD_BUFF_DATA10.RBT17_BT_CODE_NO := W#16#0;
   S701_WELD_BUFF_DATA10.RBT17_WELD_COUNT := W#16#0;
   S701_WELD_BUFF_DATA10.RBT18_BT_CODE_NO := W#16#0;
   S701_WELD_BUFF_DATA10.RBT18_WELD_COUNT := W#16#0;
   S701_WELD_BUFF_DATA10.RBT19_BT_CODE_NO := W#16#0;
   S701_WELD_BUFF_DATA10.RBT19_WELD_COUNT := W#16#0;
   S701_WELD_BUFF_DATA10.RBT20_BT_CODE_NO := W#16#0;
   S701_WELD_BUFF_DATA10.RBT20_WELD_COUNT := W#16#0;
   S701_WELD_BUFF_DATA10.RBT21_BT_CODE_NO := W#16#0;
   S701_WELD_BUFF_DATA10.RBT21_WELD_COUNT := W#16#0;
   S701_WELD_BUFF_DATA10.RBT22_BT_CODE_NO := W#16#0;
   S701_WELD_BUFF_DATA10.RBT22_WELD_COUNT := W#16#0;
   S701_WELD_BUFF_DATA10.RBT23_BT_CODE_NO := W#16#0;
   S701_WELD_BUFF_DATA10.RBT23_WELD_COUNT := W#16#0;
   S701_WELD_BUFF_DATA10.RBT24_BT_CODE_NO := W#16#0;
   S701_WELD_BUFF_DATA10.RBT24_WELD_COUNT := W#16#0;
   S701_WELD_BUFF_DATA10.WELD_DETERMINES_RESULT := W#16#0;
   S701_WELD_BUFF_DATA10.WELD_CHECK_SUM := W#16#0;
   S701_WELD_BUFF_DATA10.SPARE1 := W#16#0;
END_DATA_BLOCK

DATA_BLOCK DB 45
TITLE =
VERSION : 0.1


  STRUCT
   STAT0 : ARRAY  [0 .. 99 ] OF WORD  := W#16#0;
   STAT01 : ARRAY  [0 .. 99 ] OF WORD  := W#16#0;
   STAT02 : ARRAY  [0 .. 99 ] OF WORD  := W#16#0;
  END_STRUCT ;
BEGIN
   STAT0[0] := W#16#0;
   STAT0[1] := W#16#0;
   STAT0[2] := W#16#0;
   STAT0[3] := W#16#0;
   STAT0[4] := W#16#0;
   STAT0[5] := W#16#0;
   STAT0[6] := W#16#0;
   STAT0[7] := W#16#0;
   STAT0[8] := W#16#0;
   STAT0[9] := W#16#0;
   STAT0[10] := W#16#0;
   STAT0[11] := W#16#0;
   STAT0[12] := W#16#0;
   STAT0[13] := W#16#0;
   STAT0[14] := W#16#0;
   STAT0[15] := W#16#0;
   STAT0[16] := W#16#0;
   STAT0[17] := W#16#0;
   STAT0[18] := W#16#0;
   STAT0[19] := W#16#0;
   STAT0[20] := W#16#0;
   STAT0[21] := W#16#0;
   STAT0[22] := W#16#0;
   STAT0[23] := W#16#0;
   STAT0[24] := W#16#0;
   STAT0[25] := W#16#0;
   STAT0[26] := W#16#0;
   STAT0[27] := W#16#0;
   STAT0[28] := W#16#0;
   STAT0[29] := W#16#0;
   STAT0[30] := W#16#0;
   STAT0[31] := W#16#0;
   STAT0[32] := W#16#0;
   STAT0[33] := W#16#0;
   STAT0[34] := W#16#0;
   STAT0[35] := W#16#0;
   STAT0[36] := W#16#0;
   STAT0[37] := W#16#0;
   STAT0[38] := W#16#0;
   STAT0[39] := W#16#0;
   STAT0[40] := W#16#0;
   STAT0[41] := W#16#0;
   STAT0[42] := W#16#0;
   STAT0[43] := W#16#0;
   STAT0[44] := W#16#0;
   STAT0[45] := W#16#0;
   STAT0[46] := W#16#0;
   STAT0[47] := W#16#0;
   STAT0[48] := W#16#0;
   STAT0[49] := W#16#0;
   STAT0[50] := W#16#0;
   STAT0[51] := W#16#0;
   STAT0[52] := W#16#0;
   STAT0[53] := W#16#0;
   STAT0[54] := W#16#0;
   STAT0[55] := W#16#0;
   STAT0[56] := W#16#0;
   STAT0[57] := W#16#0;
   STAT0[58] := W#16#0;
   STAT0[59] := W#16#0;
   STAT0[60] := W#16#0;
   STAT0[61] := W#16#0;
   STAT0[62] := W#16#0;
   STAT0[63] := W#16#0;
   STAT0[64] := W#16#0;
   STAT0[65] := W#16#0;
   STAT0[66] := W#16#0;
   STAT0[67] := W#16#0;
   STAT0[68] := W#16#0;
   STAT0[69] := W#16#0;
   STAT0[70] := W#16#0;
   STAT0[71] := W#16#0;
   STAT0[72] := W#16#0;
   STAT0[73] := W#16#0;
   STAT0[74] := W#16#0;
   STAT0[75] := W#16#0;
   STAT0[76] := W#16#0;
   STAT0[77] := W#16#0;
   STAT0[78] := W#16#0;
   STAT0[79] := W#16#0;
   STAT0[80] := W#16#0;
   STAT0[81] := W#16#0;
   STAT0[82] := W#16#0;
   STAT0[83] := W#16#0;
   STAT0[84] := W#16#0;
   STAT0[85] := W#16#0;
   STAT0[86] := W#16#0;
   STAT0[87] := W#16#0;
   STAT0[88] := W#16#0;
   STAT0[89] := W#16#0;
   STAT0[90] := W#16#0;
   STAT0[91] := W#16#0;
   STAT0[92] := W#16#0;
   STAT0[93] := W#16#0;
   STAT0[94] := W#16#0;
   STAT0[95] := W#16#0;
   STAT0[96] := W#16#0;
   STAT0[97] := W#16#0;
   STAT0[98] := W#16#0;
   STAT0[99] := W#16#0;
   STAT01[0] := W#16#0;
   STAT01[1] := W#16#0;
   STAT01[2] := W#16#0;
   STAT01[3] := W#16#0;
   STAT01[4] := W#16#0;
   STAT01[5] := W#16#0;
   STAT01[6] := W#16#0;
   STAT01[7] := W#16#0;
   STAT01[8] := W#16#0;
   STAT01[9] := W#16#0;
   STAT01[10] := W#16#0;
   STAT01[11] := W#16#0;
   STAT01[12] := W#16#0;
   STAT01[13] := W#16#0;
   STAT01[14] := W#16#0;
   STAT01[15] := W#16#0;
   STAT01[16] := W#16#0;
   STAT01[17] := W#16#0;
   STAT01[18] := W#16#0;
   STAT01[19] := W#16#0;
   STAT01[20] := W#16#0;
   STAT01[21] := W#16#0;
   STAT01[22] := W#16#0;
   STAT01[23] := W#16#0;
   STAT01[24] := W#16#0;
   STAT01[25] := W#16#0;
   STAT01[26] := W#16#0;
   STAT01[27] := W#16#0;
   STAT01[28] := W#16#0;
   STAT01[29] := W#16#0;
   STAT01[30] := W#16#0;
   STAT01[31] := W#16#0;
   STAT01[32] := W#16#0;
   STAT01[33] := W#16#0;
   STAT01[34] := W#16#0;
   STAT01[35] := W#16#0;
   STAT01[36] := W#16#0;
   STAT01[37] := W#16#0;
   STAT01[38] := W#16#0;
   STAT01[39] := W#16#0;
   STAT01[40] := W#16#0;
   STAT01[41] := W#16#0;
   STAT01[42] := W#16#0;
   STAT01[43] := W#16#0;
   STAT01[44] := W#16#0;
   STAT01[45] := W#16#0;
   STAT01[46] := W#16#0;
   STAT01[47] := W#16#0;
   STAT01[48] := W#16#0;
   STAT01[49] := W#16#0;
   STAT01[50] := W#16#0;
   STAT01[51] := W#16#0;
   STAT01[52] := W#16#0;
   STAT01[53] := W#16#0;
   STAT01[54] := W#16#0;
   STAT01[55] := W#16#0;
   STAT01[56] := W#16#0;
   STAT01[57] := W#16#0;
   STAT01[58] := W#16#0;
   STAT01[59] := W#16#0;
   STAT01[60] := W#16#0;
   STAT01[61] := W#16#0;
   STAT01[62] := W#16#0;
   STAT01[63] := W#16#0;
   STAT01[64] := W#16#0;
   STAT01[65] := W#16#0;
   STAT01[66] := W#16#0;
   STAT01[67] := W#16#0;
   STAT01[68] := W#16#0;
   STAT01[69] := W#16#0;
   STAT01[70] := W#16#0;
   STAT01[71] := W#16#0;
   STAT01[72] := W#16#0;
   STAT01[73] := W#16#0;
   STAT01[74] := W#16#0;
   STAT01[75] := W#16#0;
   STAT01[76] := W#16#0;
   STAT01[77] := W#16#0;
   STAT01[78] := W#16#0;
   STAT01[79] := W#16#0;
   STAT01[80] := W#16#0;
   STAT01[81] := W#16#0;
   STAT01[82] := W#16#0;
   STAT01[83] := W#16#0;
   STAT01[84] := W#16#0;
   STAT01[85] := W#16#0;
   STAT01[86] := W#16#0;
   STAT01[87] := W#16#0;
   STAT01[88] := W#16#0;
   STAT01[89] := W#16#0;
   STAT01[90] := W#16#0;
   STAT01[91] := W#16#0;
   STAT01[92] := W#16#0;
   STAT01[93] := W#16#0;
   STAT01[94] := W#16#0;
   STAT01[95] := W#16#0;
   STAT01[96] := W#16#0;
   STAT01[97] := W#16#0;
   STAT01[98] := W#16#0;
   STAT01[99] := W#16#0;
   STAT02[0] := W#16#0;
   STAT02[1] := W#16#0;
   STAT02[2] := W#16#0;
   STAT02[3] := W#16#0;
   STAT02[4] := W#16#0;
   STAT02[5] := W#16#0;
   STAT02[6] := W#16#0;
   STAT02[7] := W#16#0;
   STAT02[8] := W#16#0;
   STAT02[9] := W#16#0;
   STAT02[10] := W#16#0;
   STAT02[11] := W#16#0;
   STAT02[12] := W#16#0;
   STAT02[13] := W#16#0;
   STAT02[14] := W#16#0;
   STAT02[15] := W#16#0;
   STAT02[16] := W#16#0;
   STAT02[17] := W#16#0;
   STAT02[18] := W#16#0;
   STAT02[19] := W#16#0;
   STAT02[20] := W#16#0;
   STAT02[21] := W#16#0;
   STAT02[22] := W#16#0;
   STAT02[23] := W#16#0;
   STAT02[24] := W#16#0;
   STAT02[25] := W#16#0;
   STAT02[26] := W#16#0;
   STAT02[27] := W#16#0;
   STAT02[28] := W#16#0;
   STAT02[29] := W#16#0;
   STAT02[30] := W#16#0;
   STAT02[31] := W#16#0;
   STAT02[32] := W#16#0;
   STAT02[33] := W#16#0;
   STAT02[34] := W#16#0;
   STAT02[35] := W#16#0;
   STAT02[36] := W#16#0;
   STAT02[37] := W#16#0;
   STAT02[38] := W#16#0;
   STAT02[39] := W#16#0;
   STAT02[40] := W#16#0;
   STAT02[41] := W#16#0;
   STAT02[42] := W#16#0;
   STAT02[43] := W#16#0;
   STAT02[44] := W#16#0;
   STAT02[45] := W#16#0;
   STAT02[46] := W#16#0;
   STAT02[47] := W#16#0;
   STAT02[48] := W#16#0;
   STAT02[49] := W#16#0;
   STAT02[50] := W#16#0;
   STAT02[51] := W#16#0;
   STAT02[52] := W#16#0;
   STAT02[53] := W#16#0;
   STAT02[54] := W#16#0;
   STAT02[55] := W#16#0;
   STAT02[56] := W#16#0;
   STAT02[57] := W#16#0;
   STAT02[58] := W#16#0;
   STAT02[59] := W#16#0;
   STAT02[60] := W#16#0;
   STAT02[61] := W#16#0;
   STAT02[62] := W#16#0;
   STAT02[63] := W#16#0;
   STAT02[64] := W#16#0;
   STAT02[65] := W#16#0;
   STAT02[66] := W#16#0;
   STAT02[67] := W#16#0;
   STAT02[68] := W#16#0;
   STAT02[69] := W#16#0;
   STAT02[70] := W#16#0;
   STAT02[71] := W#16#0;
   STAT02[72] := W#16#0;
   STAT02[73] := W#16#0;
   STAT02[74] := W#16#0;
   STAT02[75] := W#16#0;
   STAT02[76] := W#16#0;
   STAT02[77] := W#16#0;
   STAT02[78] := W#16#0;
   STAT02[79] := W#16#0;
   STAT02[80] := W#16#0;
   STAT02[81] := W#16#0;
   STAT02[82] := W#16#0;
   STAT02[83] := W#16#0;
   STAT02[84] := W#16#0;
   STAT02[85] := W#16#0;
   STAT02[86] := W#16#0;
   STAT02[87] := W#16#0;
   STAT02[88] := W#16#0;
   STAT02[89] := W#16#0;
   STAT02[90] := W#16#0;
   STAT02[91] := W#16#0;
   STAT02[92] := W#16#0;
   STAT02[93] := W#16#0;
   STAT02[94] := W#16#0;
   STAT02[95] := W#16#0;
   STAT02[96] := W#16#0;
   STAT02[97] := W#16#0;
   STAT02[98] := W#16#0;
   STAT02[99] := W#16#0;
END_DATA_BLOCK

DATA_BLOCK DB 49
TITLE =
VERSION : 0.1


  STRUCT
   OTR_PLT : STRUCT
    PLT3_ERROR : BOOL ;
    PLT4_ERROR : BOOL ;
    PLT5_ERROR : BOOL ;
    PLT6_ERROR : BOOL ;
    PLT9_ERROR : BOOL ;
    PLT10_ERROR : BOOL ;
    PLT11_ERROR : BOOL ;
    PLT12_ERROR : BOOL ;
    PLT3_BT_ERROR : BOOL ;
    PLT4_BT_ERROR : BOOL ;
    PLT5_BT_ERROR : BOOL ;
    PLT6_BT_ERROR : BOOL ;
    PLT9_BT_ERROR : BOOL ;
    PLT10_BT_ERROR : BOOL ;
    PLT11_BT_ERROR : BOOL ;
    PLT12_BT_ERROR : BOOL ;
    PLT_BT_SELECT : BOOL ;
    PLT_BT_SELECT_ON : BOOL ;
    SPARE1 : BOOL ;
    SPARE2 : BOOL ;
    SPARE3 : BOOL ;
    SPARE4 : BOOL ;
    SPARE5 : BOOL ;
    SPARE6 : BOOL ;
    PLT3_LM_SELECT : BOOL ;
    PLT3_TL_SELECT : BOOL ;
    PLT3_LM : BOOL ;
    PLT3_TL : BOOL ;
    PLT3_LM_LOAD_OK : BOOL ;
    PLT3_TL_LOAD_OK : BOOL ;
    PLT3_LM_LOAD_COMPL : BOOL ;
    PLT3_TL_LOAD_COMPL : BOOL ;
    PLT4_LM_SELECT : BOOL ;
    PLT4_TL_SELECT : BOOL ;
    PLT4_LM : BOOL ;
    PLT4_TL : BOOL ;
    PLT4_LM_LOAD_OK : BOOL ;
    PLT4_TL_LOAD_OK : BOOL ;
    PLT4_LM_LOAD_COMPL : BOOL ;
    PLT4_TL_LOAD_COMPL : BOOL ;
    PLT5_LM_SELECT : BOOL ;
    PLT5_TL_SELECT : BOOL ;
    PLT5_LM : BOOL ;
    PLT5_TL : BOOL ;
    PLT5_LM_LOAD_OK : BOOL ;
    PLT5_TL_LOAD_OK : BOOL ;
    PLT5_LM_LOAD_COMPL : BOOL ;
    PLT5_TL_LOAD_COMPL : BOOL ;
    PLT6_LM_SELECT : BOOL ;
    PLT6_TL_SELECT : BOOL ;
    PLT6_LM : BOOL ;
    PLT6_TL : BOOL ;
    PLT6_LM_LOAD_OK : BOOL ;
    PLT6_TL_LOAD_OK : BOOL ;
    PLT6_LM_LOAD_COMPL : BOOL ;
    PLT6_TL_LOAD_COMPL : BOOL ;
    SPARE7 : BOOL ;
    SPARE8 : BOOL ;
    SPARE9 : BOOL ;
    SPARE10 : BOOL ;
    SPARE11 : BOOL ;
    SPARE12 : BOOL ;
    SPARE13 : BOOL ;
    SPARE14 : BOOL ;
    SPARE15 : BOOL ;
    SPARE16 : BOOL ;
    SPARE17 : BOOL ;
    SPARE18 : BOOL ;
    SPARE19 : BOOL ;
    SPARE20 : BOOL ;
    SPARE21 : BOOL ;
    SPARE22 : BOOL ;
    PLT9_LM_SELECT : BOOL ;
    PLT9_TL_SELECT : BOOL ;
    PLT9_LM : BOOL ;
    PLT9_TL : BOOL ;
    PLT9_LM_LOAD_OK : BOOL ;
    PLT9_TL_LOAD_OK : BOOL ;
    PLT9_LM_LOAD_COMPL : BOOL ;
    PLT9_TL_LOAD_COMPL : BOOL ;
    PLT10_LM_SELECT : BOOL ;
    PLT10_TL_SELECT : BOOL ;
    PLT10_LM : BOOL ;
    PLT10_TL : BOOL ;
    PLT10_LM_LOAD_OK : BOOL ;
    PLT10_TL_LOAD_OK : BOOL ;
    PLT10_LM_LOAD_COMPL : BOOL ;
    PLT10_TL_LOAD_COMPL : BOOL ;
    PLT11_LM_SELECT : BOOL ;
    PLT11_TL_SELECT : BOOL ;
    PLT11_LM : BOOL ;
    PLT11_TL : BOOL ;
    PLT11_LM_LOAD_OK : BOOL ;
    PLT11_TL_LOAD_OK : BOOL ;
    PLT11_LM_LOAD_COMPL : BOOL ;
    PLT11_TL_LOAD_COMPL : BOOL ;
    PLT12_LM_SELECT : BOOL ;
    PLT12_TL_SELECT : BOOL ;
    PLT12_LM : BOOL ;
    PLT12_TL : BOOL ;
    PLT12_LM_LOAD_OK : BOOL ;
    PLT12_TL_LOAD_OK : BOOL ;
    PLT12_LM_LOAD_COMPL : BOOL ;
    PLT12_TL_LOAD_COMPL : BOOL ;
    SPARE23 : BOOL ;
    SPARE24 : BOOL ;
    SPARE25 : BOOL ;
    SPARE26 : BOOL ;
    SPARE27 : BOOL ;
    SPARE28 : BOOL ;
    SPARE29 : BOOL ;
    SPARE30 : BOOL ;
   END_STRUCT ;
  END_STRUCT ;
BEGIN
   OTR_PLT.PLT3_ERROR := FALSE;
   OTR_PLT.PLT4_ERROR := FALSE;
   OTR_PLT.PLT5_ERROR := FALSE;
   OTR_PLT.PLT6_ERROR := FALSE;
   OTR_PLT.PLT9_ERROR := FALSE;
   OTR_PLT.PLT10_ERROR := FALSE;
   OTR_PLT.PLT11_ERROR := FALSE;
   OTR_PLT.PLT12_ERROR := FALSE;
   OTR_PLT.PLT3_BT_ERROR := FALSE;
   OTR_PLT.PLT4_BT_ERROR := FALSE;
   OTR_PLT.PLT5_BT_ERROR := FALSE;
   OTR_PLT.PLT6_BT_ERROR := FALSE;
   OTR_PLT.PLT9_BT_ERROR := FALSE;
   OTR_PLT.PLT10_BT_ERROR := FALSE;
   OTR_PLT.PLT11_BT_ERROR := FALSE;
   OTR_PLT.PLT12_BT_ERROR := FALSE;
   OTR_PLT.PLT_BT_SELECT := FALSE;
   OTR_PLT.PLT_BT_SELECT_ON := FALSE;
   OTR_PLT.SPARE1 := FALSE;
   OTR_PLT.SPARE2 := FALSE;
   OTR_PLT.SPARE3 := FALSE;
   OTR_PLT.SPARE4 := FALSE;
   OTR_PLT.SPARE5 := FALSE;
   OTR_PLT.SPARE6 := FALSE;
   OTR_PLT.PLT3_LM_SELECT := FALSE;
   OTR_PLT.PLT3_TL_SELECT := FALSE;
   OTR_PLT.PLT3_LM := FALSE;
   OTR_PLT.PLT3_TL := FALSE;
   OTR_PLT.PLT3_LM_LOAD_OK := FALSE;
   OTR_PLT.PLT3_TL_LOAD_OK := FALSE;
   OTR_PLT.PLT3_LM_LOAD_COMPL := FALSE;
   OTR_PLT.PLT3_TL_LOAD_COMPL := FALSE;
   OTR_PLT.PLT4_LM_SELECT := FALSE;
   OTR_PLT.PLT4_TL_SELECT := FALSE;
   OTR_PLT.PLT4_LM := FALSE;
   OTR_PLT.PLT4_TL := FALSE;
   OTR_PLT.PLT4_LM_LOAD_OK := FALSE;
   OTR_PLT.PLT4_TL_LOAD_OK := FALSE;
   OTR_PLT.PLT4_LM_LOAD_COMPL := FALSE;
   OTR_PLT.PLT4_TL_LOAD_COMPL := FALSE;
   OTR_PLT.PLT5_LM_SELECT := FALSE;
   OTR_PLT.PLT5_TL_SELECT := FALSE;
   OTR_PLT.PLT5_LM := FALSE;
   OTR_PLT.PLT5_TL := FALSE;
   OTR_PLT.PLT5_LM_LOAD_OK := FALSE;
   OTR_PLT.PLT5_TL_LOAD_OK := FALSE;
   OTR_PLT.PLT5_LM_LOAD_COMPL := FALSE;
   OTR_PLT.PLT5_TL_LOAD_COMPL := FALSE;
   OTR_PLT.PLT6_LM_SELECT := FALSE;
   OTR_PLT.PLT6_TL_SELECT := FALSE;
   OTR_PLT.PLT6_LM := FALSE;
   OTR_PLT.PLT6_TL := FALSE;
   OTR_PLT.PLT6_LM_LOAD_OK := FALSE;
   OTR_PLT.PLT6_TL_LOAD_OK := FALSE;
   OTR_PLT.PLT6_LM_LOAD_COMPL := FALSE;
   OTR_PLT.PLT6_TL_LOAD_COMPL := FALSE;
   OTR_PLT.SPARE7 := FALSE;
   OTR_PLT.SPARE8 := FALSE;
   OTR_PLT.SPARE9 := FALSE;
   OTR_PLT.SPARE10 := FALSE;
   OTR_PLT.SPARE11 := FALSE;
   OTR_PLT.SPARE12 := FALSE;
   OTR_PLT.SPARE13 := FALSE;
   OTR_PLT.SPARE14 := FALSE;
   OTR_PLT.SPARE15 := FALSE;
   OTR_PLT.SPARE16 := FALSE;
   OTR_PLT.SPARE17 := FALSE;
   OTR_PLT.SPARE18 := FALSE;
   OTR_PLT.SPARE19 := FALSE;
   OTR_PLT.SPARE20 := FALSE;
   OTR_PLT.SPARE21 := FALSE;
   OTR_PLT.SPARE22 := FALSE;
   OTR_PLT.PLT9_LM_SELECT := FALSE;
   OTR_PLT.PLT9_TL_SELECT := FALSE;
   OTR_PLT.PLT9_LM := FALSE;
   OTR_PLT.PLT9_TL := FALSE;
   OTR_PLT.PLT9_LM_LOAD_OK := FALSE;
   OTR_PLT.PLT9_TL_LOAD_OK := FALSE;
   OTR_PLT.PLT9_LM_LOAD_COMPL := FALSE;
   OTR_PLT.PLT9_TL_LOAD_COMPL := FALSE;
   OTR_PLT.PLT10_LM_SELECT := FALSE;
   OTR_PLT.PLT10_TL_SELECT := FALSE;
   OTR_PLT.PLT10_LM := FALSE;
   OTR_PLT.PLT10_TL := FALSE;
   OTR_PLT.PLT10_LM_LOAD_OK := FALSE;
   OTR_PLT.PLT10_TL_LOAD_OK := FALSE;
   OTR_PLT.PLT10_LM_LOAD_COMPL := FALSE;
   OTR_PLT.PLT10_TL_LOAD_COMPL := FALSE;
   OTR_PLT.PLT11_LM_SELECT := FALSE;
   OTR_PLT.PLT11_TL_SELECT := FALSE;
   OTR_PLT.PLT11_LM := FALSE;
   OTR_PLT.PLT11_TL := FALSE;
   OTR_PLT.PLT11_LM_LOAD_OK := FALSE;
   OTR_PLT.PLT11_TL_LOAD_OK := FALSE;
   OTR_PLT.PLT11_LM_LOAD_COMPL := FALSE;
   OTR_PLT.PLT11_TL_LOAD_COMPL := FALSE;
   OTR_PLT.PLT12_LM_SELECT := FALSE;
   OTR_PLT.PLT12_TL_SELECT := FALSE;
   OTR_PLT.PLT12_LM := FALSE;
   OTR_PLT.PLT12_TL := FALSE;
   OTR_PLT.PLT12_LM_LOAD_OK := FALSE;
   OTR_PLT.PLT12_TL_LOAD_OK := FALSE;
   OTR_PLT.PLT12_LM_LOAD_COMPL := FALSE;
   OTR_PLT.PLT12_TL_LOAD_COMPL := FALSE;
   OTR_PLT.SPARE23 := FALSE;
   OTR_PLT.SPARE24 := FALSE;
   OTR_PLT.SPARE25 := FALSE;
   OTR_PLT.SPARE26 := FALSE;
   OTR_PLT.SPARE27 := FALSE;
   OTR_PLT.SPARE28 := FALSE;
   OTR_PLT.SPARE29 := FALSE;
   OTR_PLT.SPARE30 := FALSE;
END_DATA_BLOCK

DATA_BLOCK DB 51
TITLE =
VERSION : 0.1


